KUKA KRL program: f1_Kuka_APT211T02S11.SRC

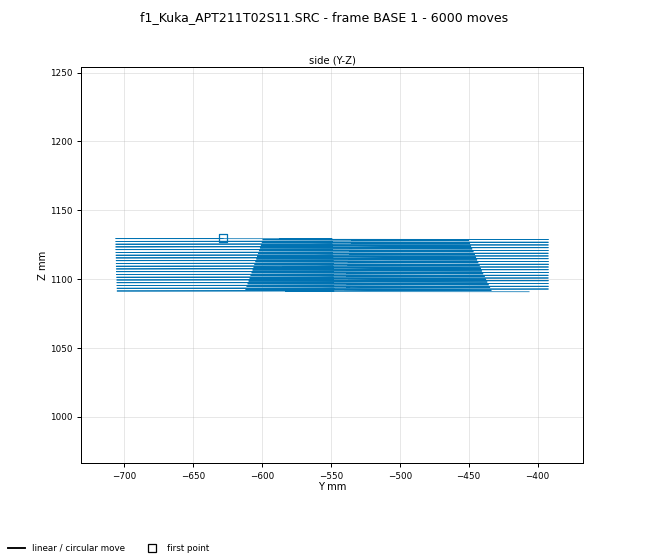
[picture p0: tool path of f1_Kuka_APT211T02S11.SRC in frame BASE 1, 6000 of 6001 moves have a stored position in this frame; points joined in program order, loops and branches not executed]
&ACCESS RVP
&REL 2
&PARAM TEMPLATE = C:\KRC\Roboter\Template\vorgabe
&PARAM EDITMASK = *
DEF f1_Kuka_APT211T02S11()


;FOLD INI;%{PE}%V3.2.0,%MKUKATPBASIS,%CINIT,%VCOMMON,%P
  ;FOLD BAS INI;%{E}%V3.2.0,%MKUKATPBASIS,%CINIT,%VINIT,%P
    GLOBAL INTERRUPT DECL 3 WHEN $STOPMESS==TRUE DO IR_STOPM ( )
    INTERRUPT ON 3
    BAS (#INITMOV,0 )
  ;ENDFOLD (BAS INI)
  ;FOLD USER INI;%{E}%V3.2.0,%MKUKATPUSER,%CINIT,%VINIT,%P
    ;Make your modifications here
  ;ENDFOLD (USER INI)
;ENDFOLD (INI)


;*** Make Null PTP Move
  PTP $pos_act

;*** Auto Load The Correct TOOL Data
  $tool=tool_data[2]

;*** Auto Load The Correct BASE Data
  $base=base_data[1]

  $ADVANCE = 5

;*** Restate Last Velocity
MMPM(30000.0)
SetRPM(8000)
LIN {X 0.276,Y -628.443,Z 1129.655,A 0.000,B 0.000,C 90.000,E1 153.896} C_DIS
LIN {X -0.160,Y -631.437,Z 1129.648,A 0.000,B 0.000,C 90.000,E1 152.666} C_DIS
LIN {X 0.011,Y -634.210,Z 1129.641,A 0.000,B 0.000,C 90.000,E1 151.385} C_DIS
LIN {X -0.027,Y -636.938,Z 1129.634,A 0.000,B 0.000,C 90.000,E1 150.127} C_DIS
LIN {X -0.018,Y -639.541,Z 1129.627,A 0.000,B 0.000,C 90.000,E1 148.869} C_DIS
LIN {X -0.027,Y -641.475,Z 1129.621,A 0.000,B 0.000,C 90.000,E1 147.867} C_DIS
LIN {X -0.154,Y -643.842,Z 1129.615,A 0.000,B 0.000,C 90.000,E1 146.628} C_DIS
LIN {X -0.238,Y -646.087,Z 1129.608,A 0.000,B 0.000,C 90.000,E1 145.388} C_DIS
LIN {X 0.084,Y -648.177,Z 1129.601,A 0.000,B 0.000,C 90.000,E1 144.116} C_DIS
LIN {X -0.031,Y -650.714,Z 1129.592,A 0.000,B 0.000,C 90.000,E1 142.637} C_DIS
LIN {X -0.300,Y -654.664,Z 1129.580,A 0.000,B 0.000,C 90.000,E1 140.436} C_DIS
LIN {X -0.032,Y -657.890,Z 1129.571,A 0.000,B 0.000,C 90.000,E1 138.690} C_DIS
LIN {X -0.154,Y -660.769,Z 1129.562,A 0.000,B 0.000,C 90.000,E1 137.229} C_DIS
LIN {X 0.211,Y -664.786,Z 1129.552,A 0.000,B 0.000,C 90.000,E1 135.243} C_DIS
LIN {X 0.204,Y -669.174,Z 1129.541,A 0.000,B 0.000,C 90.000,E1 133.299} C_DIS
LIN {X -0.116,Y -673.801,Z 1129.530,A 0.000,B 0.000,C 90.000,E1 131.391} C_DIS
LIN {X 0.050,Y -676.665,Z 1129.523,A 0.000,B 0.000,C 90.000,E1 130.172} C_DIS
LIN {X 0.038,Y -682.177,Z 1129.511,A 0.000,B 0.000,C 90.000,E1 128.016} C_DIS
LIN {X -0.141,Y -684.591,Z 1129.506,A 0.000,B 0.000,C 90.000,E1 127.076} C_DIS
LIN {X -0.113,Y -687.597,Z 1129.499,A 0.000,B 0.000,C 90.000,E1 125.884} C_DIS
LIN {X -0.232,Y -689.932,Z 1129.494,A 0.000,B 0.000,C 90.000,E1 124.945} C_DIS
LIN {X -0.261,Y -693.988,Z 1129.485,A 0.000,B 0.000,C 90.000,E1 123.293} C_DIS
LIN {X -0.123,Y -696.176,Z 1129.480,A 0.000,B 0.000,C 90.000,E1 122.339} C_DIS
LIN {X 0.292,Y -698.628,Z 1129.473,A 0.000,B 0.000,C 90.000,E1 121.131} C_DIS
LIN {X -0.135,Y -699.916,Z 1129.469,A 0.000,B 0.000,C 90.000,E1 120.463} C_DIS
LIN {X 0.203,Y -703.162,Z 1129.459,A 0.000,B 0.000,C 90.000,E1 118.565} C_DIS
LIN {X 0.147,Y -703.966,Z 1129.456,A 0.000,B 0.000,C 90.000,E1 118.103} C_DIS
LIN {X 0.378,Y -704.856,Z 1129.452,A 0.000,B 0.000,C 90.000,E1 117.385} C_DIS
LIN {X -0.043,Y -705.630,Z 1129.447,A 0.000,B 0.000,C 90.000,E1 116.488} C_DIS
LIN {X 0.182,Y -706.158,Z 1129.442,A 0.000,B 0.000,C 90.000,E1 115.540} C_DIS
LIN {X 0.128,Y -706.298,Z 1129.439,A 0.000,B 0.000,C 90.000,E1 115.079} C_DIS
LIN {X -0.226,Y -706.173,Z 1129.437,A 0.000,B 0.000,C 90.000,E1 114.643} C_DIS
LIN {X 0.066,Y -705.417,Z 1129.434,A 0.000,B 0.000,C 90.000,E1 114.155} C_DIS
LIN {X -0.288,Y -704.953,Z 1129.433,A 0.000,B 0.000,C 90.000,E1 113.951} C_DIS
LIN {X 0.000,Y -703.071,Z 1129.430,A 0.000,B 0.000,C 90.000,E1 113.462} C_DIS
LIN {X 0.281,Y -701.852,Z 1129.429,A 0.000,B 0.000,C 90.000,E1 113.206} C_DIS
LIN {X -0.094,Y -697.553,Z 1129.427,A 0.000,B 0.000,C 90.000,E1 112.770} C_DIS
LIN {X 0.035,Y -696.242,Z 1129.426,A 0.000,B 0.000,C 90.000,E1 112.642} C_DIS
LIN {X 0.163,Y -694.128,Z 1129.425,A 0.000,B 0.000,C 90.000,E1 112.514} C_DIS
LIN {X 0.381,Y -685.961,Z 1129.424,A 0.000,B 0.000,C 90.000,E1 112.206} C_DIS
LIN {X -0.097,Y -683.808,Z 1129.423,A 0.000,B 0.000,C 90.000,E1 112.206} C_DIS
LIN {X -0.315,Y -676.021,Z 1129.423,A 0.000,B 0.000,C 90.000,E1 112.153} C_DIS
LIN {X -0.314,Y -603.131,Z 1129.423,A 0.000,B 0.000,C 90.000,E1 112.153} C_DIS
LIN {X 0.332,Y -600.065,Z 1129.422,A 0.000,B 0.000,C 90.000,E1 111.897} C_DIS
LIN {X 0.084,Y -594.320,Z 1129.419,A 0.000,B 0.000,C 90.000,E1 111.461} C_DIS
LIN {X 0.254,Y -580.953,Z 1129.413,A 0.000,B 0.000,C 90.000,E1 110.248} C_DIS
LIN {X -0.197,Y -575.369,Z 1129.410,A 0.000,B 0.000,C 90.000,E1 109.812} C_DIS
LIN {X 0.116,Y -569.427,Z 1129.407,A 0.000,B 0.000,C 90.000,E1 109.322} C_DIS
LIN {X 0.032,Y -562.993,Z 1129.405,A 0.000,B 0.000,C 90.000,E1 108.906} C_DIS
LIN {X -0.161,Y -559.687,Z 1129.404,A 0.000,B 0.000,C 90.000,E1 108.725} C_DIS
LIN {X 0.065,Y -554.754,Z 1129.402,A 0.000,B 0.000,C 90.000,E1 108.417} C_DIS
LIN {X -0.112,Y -550.525,Z 1129.401,A 0.000,B 0.000,C 90.000,E1 108.109} C_DIS
LIN {X -0.149,Y -549.468,Z 1129.400,A 0.000,B 0.000,C 90.000,E1 107.928} C_DIS
LIN {X 0.332,Y -549.450,Z 1129.400,A 0.000,B 0.000,C 90.000,E1 107.873} C_DIS
LIN {X 0.089,Y -549.159,Z 1129.398,A 0.000,B 0.000,C 90.000,E1 107.583} C_DIS
LIN {X 0.132,Y -549.580,Z 1129.393,A 0.000,B 0.000,C 90.000,E1 106.677} C_DIS
LIN {X 0.156,Y -550.378,Z 1129.387,A 0.000,B 0.000,C 90.000,E1 105.552} C_DIS
LIN {X -0.172,Y -552.315,Z 1129.373,A 0.000,B 0.000,C 90.000,E1 103.063} C_DIS
LIN {X 0.140,Y -554.030,Z 1129.362,A 0.000,B 0.000,C 90.000,E1 101.074} C_DIS
LIN {X -0.191,Y -555.490,Z 1129.352,A 0.000,B 0.000,C 90.000,E1 99.434} C_DIS
LIN {X -0.135,Y -557.119,Z 1129.343,A 0.000,B 0.000,C 90.000,E1 97.757} C_DIS
LIN {X 0.026,Y -558.898,Z 1129.332,A 0.000,B 0.000,C 90.000,E1 95.796} C_DIS
LIN {X -0.037,Y -560.091,Z 1129.325,A 0.000,B 0.000,C 90.000,E1 94.416} C_DIS
LIN {X -0.085,Y -561.163,Z 1129.317,A 0.000,B 0.000,C 90.000,E1 93.037} C_DIS
LIN {X -0.149,Y -562.106,Z 1129.309,A 0.000,B 0.000,C 90.000,E1 91.661} C_DIS
LIN {X -0.001,Y -563.356,Z 1129.298,A 0.000,B 0.000,C 90.000,E1 89.714} C_DIS
LIN {X -0.039,Y -564.181,Z 1129.291,A 0.000,B 0.000,C 90.000,E1 88.339} C_DIS
LIN {X 0.194,Y -565.188,Z 1129.280,A 0.000,B 0.000,C 90.000,E1 86.388} C_DIS
LIN {X 0.242,Y -565.857,Z 1129.272,A 0.000,B 0.000,C 90.000,E1 85.008} C_DIS
LIN {X -0.005,Y -566.679,Z 1129.262,A 0.000,B 0.000,C 90.000,E1 83.109} C_DIS
LIN {X 0.122,Y -567.264,Z 1129.254,A 0.000,B 0.000,C 90.000,E1 81.724} C_DIS
LIN {X -0.041,Y -567.961,Z 1129.245,A 0.000,B 0.000,C 90.000,E1 80.095} C_DIS
LIN {X 0.175,Y -568.982,Z 1129.233,A 0.000,B 0.000,C 90.000,E1 77.881} C_DIS
LIN {X 0.105,Y -569.580,Z 1129.225,A 0.000,B 0.000,C 90.000,E1 76.520} C_DIS
LIN {X -0.317,Y -570.930,Z 1129.212,A 0.000,B 0.000,C 90.000,E1 74.102} C_DIS
LIN {X 0.136,Y -572.366,Z 1129.199,A 0.000,B 0.000,C 90.000,E1 71.873} C_DIS
LIN {X 0.092,Y -574.123,Z 1129.187,A 0.000,B 0.000,C 90.000,E1 69.699} C_DIS
LIN {X 0.119,Y -575.359,Z 1129.180,A 0.000,B 0.000,C 90.000,E1 68.337} C_DIS
LIN {X 0.174,Y -576.690,Z 1129.172,A 0.000,B 0.000,C 90.000,E1 66.975} C_DIS
LIN {X -0.052,Y -578.301,Z 1129.162,A 0.000,B 0.000,C 90.000,E1 65.101} C_DIS
LIN {X -0.246,Y -579.488,Z 1129.154,A 0.000,B 0.000,C 90.000,E1 63.768} C_DIS
LIN {X 0.216,Y -580.828,Z 1129.145,A 0.000,B 0.000,C 90.000,E1 62.103} C_DIS
LIN {X -0.041,Y -582.020,Z 1129.136,A 0.000,B 0.000,C 90.000,E1 60.511} C_DIS
LIN {X 0.213,Y -582.736,Z 1129.130,A 0.000,B 0.000,C 90.000,E1 59.410} C_DIS
LIN {X 0.297,Y -583.784,Z 1129.121,A 0.000,B 0.000,C 90.000,E1 57.788} C_DIS
LIN {X 0.096,Y -584.829,Z 1129.111,A 0.000,B 0.000,C 90.000,E1 55.928} C_DIS
LIN {X 0.169,Y -585.420,Z 1129.105,A 0.000,B 0.000,C 90.000,E1 54.848} C_DIS
LIN {X -0.150,Y -586.436,Z 1129.094,A 0.000,B 0.000,C 90.000,E1 53.004} C_DIS
LIN {X -0.115,Y -586.917,Z 1129.087,A 0.000,B 0.000,C 90.000,E1 51.662} C_DIS
LIN {X -0.170,Y -587.342,Z 1129.081,A 0.000,B 0.000,C 90.000,E1 50.598} C_DIS
LIN {X -0.117,Y -587.578,Z 1129.074,A 0.000,B 0.000,C 90.000,E1 49.256} C_DIS
LIN {X 0.137,Y -587.582,Z 1129.068,A 0.000,B 0.000,C 90.000,E1 48.162} C_DIS
LIN {X -0.099,Y -587.323,Z 1129.059,A 0.000,B 0.000,C 90.000,E1 46.581} C_DIS
LIN {X -0.090,Y -586.888,Z 1129.051,A 0.000,B 0.000,C 90.000,E1 45.243} C_DIS
LIN {X -0.262,Y -586.375,Z 1129.045,A 0.000,B 0.000,C 90.000,E1 44.190} C_DIS
LIN {X -0.191,Y -585.866,Z 1129.041,A 0.000,B 0.000,C 90.000,E1 43.380} C_DIS
LIN {X -0.272,Y -585.528,Z 1129.038,A 0.000,B 0.000,C 90.000,E1 42.852} C_DIS
LIN {X 0.133,Y -584.133,Z 1129.031,A 0.000,B 0.000,C 90.000,E1 41.472} C_DIS
LIN {X -0.042,Y -582.853,Z 1129.025,A 0.000,B 0.000,C 90.000,E1 40.415} C_DIS
LIN {X 0.040,Y -581.798,Z 1129.020,A 0.000,B 0.000,C 90.000,E1 39.600} C_DIS
LIN {X -0.170,Y -580.155,Z 1129.014,A 0.000,B 0.000,C 90.000,E1 38.543} C_DIS
LIN {X 0.204,Y -577.753,Z 1129.007,A 0.000,B 0.000,C 90.000,E1 37.156} C_DIS
LIN {X -0.125,Y -575.914,Z 1129.002,A 0.000,B 0.000,C 90.000,E1 36.377} C_DIS
LIN {X 0.331,Y -573.866,Z 1128.998,A 0.000,B 0.000,C 90.000,E1 35.518} C_DIS
LIN {X -0.179,Y -572.343,Z 1128.995,A 0.000,B 0.000,C 90.000,E1 35.025} C_DIS
LIN {X 0.035,Y -568.837,Z 1128.989,A 0.000,B 0.000,C 90.000,E1 33.913} C_DIS
LIN {X 0.082,Y -565.703,Z 1128.984,A 0.000,B 0.000,C 90.000,E1 33.086} C_DIS
LIN {X 0.094,Y -562.230,Z 1128.979,A 0.000,B 0.000,C 90.000,E1 32.260} C_DIS
LIN {X -0.212,Y -560.378,Z 1128.977,A 0.000,B 0.000,C 90.000,E1 31.878} C_DIS
LIN {X 0.213,Y -556.350,Z 1128.972,A 0.000,B 0.000,C 90.000,E1 31.003} C_DIS
LIN {X 0.057,Y -553.399,Z 1128.969,A 0.000,B 0.000,C 90.000,E1 30.463} C_DIS
LIN {X 0.121,Y -548.863,Z 1128.965,A 0.000,B 0.000,C 90.000,E1 29.617} C_DIS
LIN {X -0.212,Y -544.695,Z 1128.961,A 0.000,B 0.000,C 90.000,E1 28.949} C_DIS
LIN {X -0.107,Y -540.200,Z 1128.957,A 0.000,B 0.000,C 90.000,E1 28.231} C_DIS
LIN {X -0.044,Y -535.300,Z 1128.953,A 0.000,B 0.000,C 90.000,E1 27.513} C_DIS
LIN {X -0.032,Y -529.995,Z 1128.949,A 0.000,B 0.000,C 90.000,E1 26.796} C_DIS
LIN {X -0.151,Y -525.471,Z 1128.946,A 0.000,B 0.000,C 90.000,E1 26.232} C_DIS
LIN {X 0.118,Y -518.189,Z 1128.941,A 0.000,B 0.000,C 90.000,E1 25.335} C_DIS
LIN {X -0.146,Y -511.760,Z 1128.937,A 0.000,B 0.000,C 90.000,E1 24.643} C_DIS
LIN {X -0.046,Y -501.108,Z 1128.931,A 0.000,B 0.000,C 90.000,E1 23.515} C_DIS
LIN {X -0.219,Y -491.482,Z 1128.925,A 0.000,B 0.000,C 90.000,E1 22.589} C_DIS
LIN {X 0.230,Y -481.334,Z 1128.920,A 0.000,B 0.000,C 90.000,E1 21.589} C_DIS
LIN {X -0.214,Y -469.631,Z 1128.914,A 0.000,B 0.000,C 90.000,E1 20.610} C_DIS
LIN {X 0.057,Y -459.552,Z 1128.909,A 0.000,B 0.000,C 90.000,E1 19.685} C_DIS
LIN {X 0.000,Y -439.216,Z 1128.899,A 0.000,B 0.000,C 90.000,E1 17.819} C_DIS
LIN {X -0.060,Y -424.920,Z 1128.891,A 0.000,B 0.000,C 90.000,E1 16.370} C_DIS
LIN {X -0.192,Y -413.778,Z 1128.884,A 0.000,B 0.000,C 90.000,E1 15.134} C_DIS
LIN {X -0.059,Y -404.421,Z 1128.877,A 0.000,B 0.000,C 90.000,E1 13.939} C_DIS
LIN {X 0.035,Y -399.506,Z 1128.874,A 0.000,B 0.000,C 90.000,E1 13.244} C_DIS
LIN {X 0.011,Y -396.631,Z 1128.871,A 0.000,B 0.000,C 90.000,E1 12.771} C_DIS
LIN {X -0.041,Y -393.975,Z 1128.868,A 0.000,B 0.000,C 90.000,E1 12.187} C_DIS
LIN {X -0.016,Y -393.344,Z 1128.867,A 0.000,B 0.000,C 90.000,E1 12.007} C_DIS
LIN {X -0.132,Y -392.375,Z 1128.865,A 0.000,B 0.000,C 90.000,E1 11.658} C_DIS
LIN {X -0.158,Y -392.079,Z 1128.862,A 0.000,B 0.000,C 90.000,E1 11.130} C_DIS
LIN {X 0.147,Y -392.624,Z 1128.859,A 0.000,B 0.000,C 90.000,E1 10.546} C_DIS
LIN {X 0.104,Y -393.154,Z 1128.857,A 0.000,B 0.000,C 90.000,E1 10.197} C_DIS
LIN {X 0.021,Y -394.627,Z 1128.853,A 0.000,B 0.000,C 90.000,E1 9.500} C_DIS
LIN {X 0.161,Y -402.489,Z 1128.837,A 0.000,B 0.000,C 90.000,E1 6.663} C_DIS
LIN {X 0.143,Y -404.784,Z 1128.833,A 0.000,B 0.000,C 90.000,E1 5.967} C_DIS
LIN {X 0.033,Y -407.437,Z 1128.830,A 0.000,B 0.000,C 90.000,E1 5.391} C_DIS
LIN {X -0.183,Y -411.799,Z 1128.827,A 0.000,B 0.000,C 90.000,E1 4.816} C_DIS
LIN {X -0.014,Y -417.173,Z 1128.824,A 0.000,B 0.000,C 90.000,E1 4.359} C_DIS
LIN {X 0.006,Y -434.964,Z 1128.817,A 0.000,B 0.000,C 90.000,E1 3.094} C_DIS
LIN {X 0.033,Y -459.488,Z 1128.808,A 0.000,B 0.000,C 90.000,E1 1.432} C_DIS
LIN {X -0.093,Y -467.649,Z 1128.805,A 0.000,B 0.000,C 90.000,E1 0.917} C_DIS
LIN {X -0.004,Y -478.874,Z 1128.801,A 0.000,B 0.000,C 90.000,E1 0.172} C_DIS
LIN {X -0.194,Y -489.209,Z 1128.797,A 0.000,B 0.000,C 90.000,E1 359.484} C_DIS
LIN {X -0.158,Y -498.343,Z 1128.793,A 0.000,B 0.000,C 90.000,E1 358.797} C_DIS
LIN {X -0.226,Y -502.919,Z 1128.791,A 0.000,B 0.000,C 90.000,E1 358.453} C_DIS
LIN {X -0.004,Y -510.065,Z 1128.788,A 0.000,B 0.000,C 90.000,E1 357.822} C_DIS
LIN {X -0.067,Y -517.099,Z 1128.784,A 0.000,B 0.000,C 90.000,E1 357.192} C_DIS
LIN {X -0.231,Y -522.381,Z 1128.781,A 0.000,B 0.000,C 90.000,E1 356.674} C_DIS
LIN {X 0.171,Y -526.361,Z 1128.779,A 0.000,B 0.000,C 90.000,E1 356.216} C_DIS
LIN {X -0.037,Y -532.551,Z 1128.775,A 0.000,B 0.000,C 90.000,E1 355.527} C_DIS
LIN {X 0.238,Y -538.039,Z 1128.771,A 0.000,B 0.000,C 90.000,E1 354.780} C_DIS
LIN {X -0.248,Y -542.168,Z 1128.768,A 0.000,B 0.000,C 90.000,E1 354.261} C_DIS
LIN {X 0.111,Y -546.634,Z 1128.764,A 0.000,B 0.000,C 90.000,E1 353.514} C_DIS
LIN {X 0.035,Y -550.776,Z 1128.760,A 0.000,B 0.000,C 90.000,E1 352.818} C_DIS
LIN {X 0.179,Y -553.798,Z 1128.757,A 0.000,B 0.000,C 90.000,E1 352.243} C_DIS
LIN {X -0.209,Y -556.605,Z 1128.754,A 0.000,B 0.000,C 90.000,E1 351.724} C_DIS
LIN {X -0.196,Y -559.702,Z 1128.750,A 0.000,B 0.000,C 90.000,E1 351.027} C_DIS
LIN {X 0.245,Y -563.057,Z 1128.745,A 0.000,B 0.000,C 90.000,E1 350.151} C_DIS
LIN {X -0.093,Y -565.111,Z 1128.742,A 0.000,B 0.000,C 90.000,E1 349.634} C_DIS
LIN {X -0.147,Y -568.067,Z 1128.738,A 0.000,B 0.000,C 90.000,E1 348.814} C_DIS
LIN {X 0.021,Y -571.609,Z 1128.732,A 0.000,B 0.000,C 90.000,E1 347.701} C_DIS
LIN {X 0.238,Y -574.908,Z 1128.726,A 0.000,B 0.000,C 90.000,E1 346.589} C_DIS
LIN {X 0.077,Y -577.993,Z 1128.720,A 0.000,B 0.000,C 90.000,E1 345.519} C_DIS
LIN {X 0.183,Y -581.645,Z 1128.712,A 0.000,B 0.000,C 90.000,E1 344.157} C_DIS
LIN {X -0.108,Y -583.762,Z 1128.708,A 0.000,B 0.000,C 90.000,E1 343.378} C_DIS
LIN {X 0.259,Y -587.109,Z 1128.700,A 0.000,B 0.000,C 90.000,E1 342.000} C_DIS
LIN {X -0.114,Y -589.570,Z 1128.694,A 0.000,B 0.000,C 90.000,E1 340.967} C_DIS
LIN {X 0.102,Y -591.882,Z 1128.688,A 0.000,B 0.000,C 90.000,E1 339.880} C_DIS
LIN {X 0.232,Y -594.457,Z 1128.681,A 0.000,B 0.000,C 90.000,E1 338.539} C_DIS
LIN {X 0.030,Y -595.433,Z 1128.678,A 0.000,B 0.000,C 90.000,E1 338.028} C_DIS
LIN {X 0.071,Y -596.576,Z 1128.674,A 0.000,B 0.000,C 90.000,E1 337.230} C_DIS
LIN {X -0.053,Y -598.137,Z 1128.666,A 0.000,B 0.000,C 90.000,E1 335.921} C_DIS
LIN {X 0.173,Y -599.005,Z 1128.660,A 0.000,B 0.000,C 90.000,E1 334.845} C_DIS
LIN {X -0.054,Y -599.388,Z 1128.656,A 0.000,B 0.000,C 90.000,E1 334.076} C_DIS
LIN {X 0.262,Y -599.490,Z 1128.652,A 0.000,B 0.000,C 90.000,E1 333.256} C_DIS
LIN {X -0.037,Y -599.218,Z 1128.646,A 0.000,B 0.000,C 90.000,E1 332.231} C_DIS
LIN {X 0.018,Y -598.634,Z 1128.641,A 0.000,B 0.000,C 90.000,E1 331.435} C_DIS
LIN {X -0.139,Y -598.037,Z 1128.638,A 0.000,B 0.000,C 90.000,E1 330.923} C_DIS
LIN {X -0.092,Y -596.865,Z 1128.634,A 0.000,B 0.000,C 90.000,E1 330.127} C_DIS
LIN {X -0.055,Y -595.245,Z 1128.630,A 0.000,B 0.000,C 90.000,E1 329.331} C_DIS
LIN {X -0.037,Y -593.230,Z 1128.625,A 0.000,B 0.000,C 90.000,E1 328.535} C_DIS
LIN {X -0.141,Y -592.478,Z 1128.624,A 0.000,B 0.000,C 90.000,E1 328.280} C_DIS
LIN {X 0.156,Y -589.637,Z 1128.619,A 0.000,B 0.000,C 90.000,E1 327.454} C_DIS
LIN {X -0.386,Y -586.404,Z 1128.615,A 0.000,B 0.000,C 90.000,E1 326.707} C_DIS
LIN {X -0.076,Y -583.355,Z 1128.611,A 0.000,B 0.000,C 90.000,E1 326.008} C_DIS
LIN {X 0.202,Y -579.925,Z 1128.607,A 0.000,B 0.000,C 90.000,E1 325.308} C_DIS
LIN {X 0.201,Y -576.931,Z 1128.604,A 0.000,B 0.000,C 90.000,E1 324.769} C_DIS
LIN {X -0.006,Y -570.210,Z 1128.598,A 0.000,B 0.000,C 90.000,E1 323.703} C_DIS
LIN {X 0.159,Y -565.536,Z 1128.595,A 0.000,B 0.000,C 90.000,E1 323.004} C_DIS
LIN {X -0.095,Y -557.371,Z 1128.589,A 0.000,B 0.000,C 90.000,E1 321.949} C_DIS
LIN {X 0.062,Y -549.505,Z 1128.583,A 0.000,B 0.000,C 90.000,E1 320.964} C_DIS
LIN {X 0.174,Y -537.721,Z 1128.575,A 0.000,B 0.000,C 90.000,E1 319.542} C_DIS
LIN {X -0.223,Y -535.682,Z 1128.574,A 0.000,B 0.000,C 90.000,E1 319.299} C_DIS
LIN {X 0.123,Y -532.461,Z 1128.571,A 0.000,B 0.000,C 90.000,E1 318.690} C_DIS
LIN {X -0.060,Y -531.568,Z 1128.570,A 0.000,B 0.000,C 90.000,E1 318.566} C_DIS
LIN {X 0.109,Y -530.858,Z 1128.569,A 0.000,B 0.000,C 90.000,E1 318.405} C_DIS
LIN {X -0.199,Y -530.175,Z 1128.568,A 0.000,B 0.000,C 90.000,E1 318.243} C_DIS
LIN {X -0.059,Y -528.452,Z 1128.566,A 0.000,B 0.000,C 90.000,E1 317.796} C_DIS
LIN {X -0.160,Y -526.830,Z 1128.562,A 0.000,B 0.000,C 90.000,E1 317.229} C_DIS
LIN {X -0.043,Y -526.104,Z 1128.560,A 0.000,B 0.000,C 90.000,E1 316.782} C_DIS
LIN {X 0.155,Y -525.395,Z 1128.555,A 0.000,B 0.000,C 90.000,E1 315.891} C_DIS
LIN {X 0.037,Y -525.202,Z 1128.552,A 0.000,B 0.000,C 90.000,E1 315.324} C_DIS
LIN {X 0.105,Y -524.824,Z 1128.544,A 0.000,B 0.000,C 90.000,E1 313.866} C_DIS
LIN {X -0.117,Y -525.254,Z 1128.528,A 0.000,B 0.000,C 90.000,E1 310.987} C_DIS
LIN {X -0.140,Y -526.429,Z 1128.515,A 0.000,B 0.000,C 90.000,E1 308.669} C_DIS
LIN {X 0.003,Y -527.504,Z 1128.505,A 0.000,B 0.000,C 90.000,E1 306.916} C_DIS
LIN {X -0.032,Y -528.643,Z 1128.495,A 0.000,B 0.000,C 90.000,E1 305.185} C_DIS
LIN {X -0.126,Y -529.510,Z 1128.489,A 0.000,B 0.000,C 90.000,E1 304.040} C_DIS
LIN {X 0.022,Y -530.997,Z 1128.478,A 0.000,B 0.000,C 90.000,E1 302.005} C_DIS
LIN {X 0.229,Y -532.317,Z 1128.468,A 0.000,B 0.000,C 90.000,E1 300.256} C_DIS
LIN {X 0.044,Y -533.168,Z 1128.462,A 0.000,B 0.000,C 90.000,E1 299.127} C_DIS
LIN {X 0.083,Y -533.934,Z 1128.456,A 0.000,B 0.000,C 90.000,E1 297.975} C_DIS
LIN {X 0.144,Y -534.499,Z 1128.449,A 0.000,B 0.000,C 90.000,E1 296.821} C_DIS
LIN {X -0.269,Y -534.874,Z 1128.443,A 0.000,B 0.000,C 90.000,E1 295.720} C_DIS
LIN {X 0.281,Y -534.998,Z 1128.436,A 0.000,B 0.000,C 90.000,E1 294.515} C_DIS
LIN {X 0.124,Y -535.054,Z 1128.430,A 0.000,B 0.000,C 90.000,E1 293.387} C_DIS
LIN {X -0.031,Y -535.106,Z 1128.422,A 0.000,B 0.000,C 90.000,E1 291.972} C_DIS
LIN {X 0.028,Y -534.993,Z 1128.413,A 0.000,B 0.000,C 90.000,E1 290.248} C_DIS
LIN {X -0.137,Y -534.782,Z 1128.405,A 0.000,B 0.000,C 90.000,E1 288.833} C_DIS
LIN {X -0.144,Y -534.430,Z 1128.397,A 0.000,B 0.000,C 90.000,E1 287.402} C_DIS
LIN {X -0.186,Y -534.064,Z 1128.390,A 0.000,B 0.000,C 90.000,E1 286.260} C_DIS
LIN {X -0.158,Y -533.295,Z 1128.381,A 0.000,B 0.000,C 90.000,E1 284.537} C_DIS
LIN {X 0.194,Y -532.589,Z 1128.373,A 0.000,B 0.000,C 90.000,E1 283.063} C_DIS
LIN {X -0.056,Y -531.688,Z 1128.363,A 0.000,B 0.000,C 90.000,E1 281.366} C_DIS
LIN {X 0.191,Y -530.743,Z 1128.354,A 0.000,B 0.000,C 90.000,E1 279.613} C_DIS
LIN {X -0.280,Y -529.834,Z 1128.344,A 0.000,B 0.000,C 90.000,E1 277.936} C_DIS
LIN {X -0.223,Y -528.819,Z 1128.333,A 0.000,B 0.000,C 90.000,E1 275.910} C_DIS
LIN {X 0.236,Y -528.209,Z 1128.325,A 0.000,B 0.000,C 90.000,E1 274.416} C_DIS
LIN {X 0.156,Y -527.568,Z 1128.317,A 0.000,B 0.000,C 90.000,E1 272.980} C_DIS
LIN {X 0.004,Y -526.806,Z 1128.307,A 0.000,B 0.000,C 90.000,E1 271.260} C_DIS
LIN {X -0.171,Y -525.989,Z 1128.297,A 0.000,B 0.000,C 90.000,E1 269.542} C_DIS
LIN {X 0.225,Y -525.480,Z 1128.291,A 0.000,B 0.000,C 90.000,E1 268.339} C_DIS
LIN {X 0.061,Y -524.748,Z 1128.283,A 0.000,B 0.000,C 90.000,E1 266.906} C_DIS
LIN {X -0.086,Y -523.713,Z 1128.273,A 0.000,B 0.000,C 90.000,E1 265.179} C_DIS
LIN {X -0.241,Y -522.938,Z 1128.267,A 0.000,B 0.000,C 90.000,E1 264.033} C_DIS
LIN {X 0.150,Y -521.520,Z 1128.259,A 0.000,B 0.000,C 90.000,E1 262.534} C_DIS
LIN {X 0.071,Y -520.126,Z 1128.251,A 0.000,B 0.000,C 90.000,E1 261.084} C_DIS
LIN {X -0.033,Y -518.715,Z 1128.242,A 0.000,B 0.000,C 90.000,E1 259.634} C_DIS
LIN {X -0.071,Y -517.334,Z 1128.234,A 0.000,B 0.000,C 90.000,E1 258.173} C_DIS
LIN {X -0.057,Y -515.314,Z 1128.223,A 0.000,B 0.000,C 90.000,E1 256.117} C_DIS
LIN {X 0.085,Y -514.002,Z 1128.215,A 0.000,B 0.000,C 90.000,E1 254.629} C_DIS
LIN {X 0.165,Y -512.216,Z 1128.205,A 0.000,B 0.000,C 90.000,E1 252.851} C_DIS
LIN {X -0.041,Y -511.026,Z 1128.198,A 0.000,B 0.000,C 90.000,E1 251.692} C_DIS
LIN {X 0.061,Y -509.782,Z 1128.192,A 0.000,B 0.000,C 90.000,E1 250.496} C_DIS
LIN {X -0.071,Y -508.118,Z 1128.183,A 0.000,B 0.000,C 90.000,E1 249.028} C_DIS
LIN {X -0.045,Y -506.433,Z 1128.175,A 0.000,B 0.000,C 90.000,E1 247.539} C_DIS
LIN {X -0.136,Y -504.926,Z 1128.169,A 0.000,B 0.000,C 90.000,E1 246.357} C_DIS
LIN {X -0.045,Y -503.360,Z 1128.162,A 0.000,B 0.000,C 90.000,E1 245.153} C_DIS
LIN {X 0.096,Y -501.199,Z 1128.154,A 0.000,B 0.000,C 90.000,E1 243.640} C_DIS
LIN {X 0.123,Y -499.434,Z 1128.147,A 0.000,B 0.000,C 90.000,E1 242.436} C_DIS
LIN {X 0.191,Y -497.098,Z 1128.139,A 0.000,B 0.000,C 90.000,E1 240.923} C_DIS
LIN {X 0.219,Y -494.663,Z 1128.130,A 0.000,B 0.000,C 90.000,E1 239.410} C_DIS
LIN {X 0.293,Y -491.602,Z 1128.120,A 0.000,B 0.000,C 90.000,E1 237.582} C_DIS
LIN {X 0.051,Y -489.060,Z 1128.112,A 0.000,B 0.000,C 90.000,E1 236.087} C_DIS
LIN {X -0.140,Y -485.944,Z 1128.101,A 0.000,B 0.000,C 90.000,E1 234.276} C_DIS
LIN {X 0.057,Y -483.240,Z 1128.093,A 0.000,B 0.000,C 90.000,E1 232.718} C_DIS
LIN {X 0.001,Y -481.107,Z 1128.086,A 0.000,B 0.000,C 90.000,E1 231.492} C_DIS
LIN {X 0.120,Y -477.710,Z 1128.076,A 0.000,B 0.000,C 90.000,E1 229.622} C_DIS
LIN {X 0.121,Y -474.327,Z 1128.065,A 0.000,B 0.000,C 90.000,E1 227.757} C_DIS
LIN {X 0.139,Y -470.398,Z 1128.053,A 0.000,B 0.000,C 90.000,E1 225.567} C_DIS
LIN {X -0.141,Y -465.834,Z 1128.038,A 0.000,B 0.000,C 90.000,E1 222.771} C_DIS
LIN {X 0.043,Y -462.152,Z 1128.024,A 0.000,B 0.000,C 90.000,E1 220.216} C_DIS
LIN {X 0.093,Y -459.617,Z 1128.013,A 0.000,B 0.000,C 90.000,E1 218.302} C_DIS
LIN {X -0.095,Y -457.023,Z 1128.000,A 0.000,B 0.000,C 90.000,E1 216.091} C_DIS
LIN {X 0.295,Y -454.845,Z 1127.990,A 0.000,B 0.000,C 90.000,E1 214.119} C_DIS
LIN {X 0.202,Y -451.679,Z 1127.970,A 0.000,B 0.000,C 90.000,E1 210.590} C_DIS
LIN {X -0.051,Y -449.938,Z 1127.949,A 0.000,B 0.000,C 90.000,E1 206.744} C_DIS
LIN {X -0.278,Y -450.279,Z 1127.940,A 0.000,B 0.000,C 90.000,E1 205.155} C_DIS
LIN {X 0.027,Y -451.189,Z 1127.932,A 0.000,B 0.000,C 90.000,E1 203.823} C_DIS
LIN {X 0.099,Y -452.383,Z 1127.927,A 0.000,B 0.000,C 90.000,E1 202.845} C_DIS
LIN {X 0.056,Y -455.799,Z 1127.916,A 0.000,B 0.000,C 90.000,E1 200.918} C_DIS
LIN {X 0.005,Y -459.488,Z 1127.907,A 0.000,B 0.000,C 90.000,E1 199.322} C_DIS
LIN {X 0.017,Y -466.025,Z 1127.895,A 0.000,B 0.000,C 90.000,E1 197.094} C_DIS
LIN {X -0.103,Y -474.605,Z 1127.881,A 0.000,B 0.000,C 90.000,E1 194.592} C_DIS
LIN {X 0.013,Y -486.289,Z 1127.864,A 0.000,B 0.000,C 90.000,E1 191.478} C_DIS
LIN {X 0.194,Y -494.854,Z 1127.852,A 0.000,B 0.000,C 90.000,E1 189.321} C_DIS
LIN {X 0.168,Y -501.028,Z 1127.844,A 0.000,B 0.000,C 90.000,E1 187.814} C_DIS
LIN {X -0.247,Y -505.941,Z 1127.837,A 0.000,B 0.000,C 90.000,E1 186.663} C_DIS
LIN {X -0.138,Y -511.919,Z 1127.829,A 0.000,B 0.000,C 90.000,E1 185.163} C_DIS
LIN {X 0.113,Y -516.758,Z 1127.822,A 0.000,B 0.000,C 90.000,E1 183.955} C_DIS
LIN {X -0.219,Y -524.051,Z 1127.812,A 0.000,B 0.000,C 90.000,E1 182.236} C_DIS
LIN {X -0.140,Y -531.802,Z 1127.802,A 0.000,B 0.000,C 90.000,E1 180.344} C_DIS
LIN {X -0.164,Y -536.667,Z 1127.796,A 0.000,B 0.000,C 90.000,E1 179.198} C_DIS
LIN {X 0.195,Y -543.296,Z 1127.787,A 0.000,B 0.000,C 90.000,E1 177.593} C_DIS
LIN {X 0.228,Y -551.080,Z 1127.777,A 0.000,B 0.000,C 90.000,E1 175.755} C_DIS
LIN {X -0.065,Y -558.889,Z 1127.766,A 0.000,B 0.000,C 90.000,E1 173.970} C_DIS
LIN {X 0.209,Y -567.288,Z 1127.756,A 0.000,B 0.000,C 90.000,E1 172.008} C_DIS
LIN {X 0.000,Y -574.375,Z 1127.747,A 0.000,B 0.000,C 90.000,E1 170.387} C_DIS
LIN {X -0.198,Y -580.103,Z 1127.739,A 0.000,B 0.000,C 90.000,E1 169.050} C_DIS
LIN {X -0.190,Y -585.565,Z 1127.732,A 0.000,B 0.000,C 90.000,E1 167.701} C_DIS
LIN {X -0.085,Y -590.948,Z 1127.724,A 0.000,B 0.000,C 90.000,E1 166.353} C_DIS
LIN {X 0.252,Y -596.015,Z 1127.717,A 0.000,B 0.000,C 90.000,E1 164.991} C_DIS
LIN {X 0.103,Y -598.873,Z 1127.712,A 0.000,B 0.000,C 90.000,E1 164.212} C_DIS
LIN {X 0.282,Y -602.430,Z 1127.707,A 0.000,B 0.000,C 90.000,E1 163.142} C_DIS
LIN {X -0.161,Y -606.719,Z 1127.699,A 0.000,B 0.000,C 90.000,E1 161.873} C_DIS
LIN {X 0.042,Y -610.721,Z 1127.692,A 0.000,B 0.000,C 90.000,E1 160.550} C_DIS
LIN {X -0.017,Y -613.792,Z 1127.686,A 0.000,B 0.000,C 90.000,E1 159.518} C_DIS
LIN {X -0.075,Y -617.327,Z 1127.679,A 0.000,B 0.000,C 90.000,E1 158.230} C_DIS
LIN {X 0.151,Y -621.444,Z 1127.671,A 0.000,B 0.000,C 90.000,E1 156.666} C_DIS
LIN {X -0.105,Y -624.680,Z 1127.663,A 0.000,B 0.000,C 90.000,E1 155.409} C_DIS
LIN {X -0.314,Y -627.838,Z 1127.656,A 0.000,B 0.000,C 90.000,E1 154.152} C_DIS
LIN {X -0.202,Y -630.870,Z 1127.649,A 0.000,B 0.000,C 90.000,E1 152.871} C_DIS
LIN {X -0.111,Y -632.572,Z 1127.645,A 0.000,B 0.000,C 90.000,E1 152.103} C_DIS
LIN {X -0.138,Y -635.866,Z 1127.637,A 0.000,B 0.000,C 90.000,E1 150.589} C_DIS
LIN {X -0.147,Y -638.504,Z 1127.630,A 0.000,B 0.000,C 90.000,E1 149.331} C_DIS
LIN {X -0.167,Y -640.540,Z 1127.624,A 0.000,B 0.000,C 90.000,E1 148.329} C_DIS
LIN {X -0.253,Y -643.369,Z 1127.616,A 0.000,B 0.000,C 90.000,E1 146.834} C_DIS
LIN {X -0.346,Y -645.624,Z 1127.609,A 0.000,B 0.000,C 90.000,E1 145.595} C_DIS
LIN {X -0.031,Y -647.756,Z 1127.602,A 0.000,B 0.000,C 90.000,E1 144.322} C_DIS
LIN {X -0.150,Y -650.297,Z 1127.594,A 0.000,B 0.000,C 90.000,E1 142.844} C_DIS
LIN {X 0.080,Y -654.237,Z 1127.581,A 0.000,B 0.000,C 90.000,E1 140.598} C_DIS
LIN {X -0.123,Y -656.980,Z 1127.573,A 0.000,B 0.000,C 90.000,E1 139.138} C_DIS
LIN {X 0.203,Y -660.334,Z 1127.563,A 0.000,B 0.000,C 90.000,E1 137.391} C_DIS
LIN {X 0.079,Y -664.818,Z 1127.551,A 0.000,B 0.000,C 90.000,E1 135.202} C_DIS
LIN {X 0.092,Y -669.805,Z 1127.539,A 0.000,B 0.000,C 90.000,E1 133.014} C_DIS
LIN {X 0.226,Y -673.866,Z 1127.530,A 0.000,B 0.000,C 90.000,E1 131.310} C_DIS
LIN {X 0.392,Y -676.737,Z 1127.523,A 0.000,B 0.000,C 90.000,E1 130.092} C_DIS
LIN {X -0.037,Y -682.266,Z 1127.511,A 0.000,B 0.000,C 90.000,E1 127.971} C_DIS
LIN {X 0.175,Y -684.128,Z 1127.507,A 0.000,B 0.000,C 90.000,E1 127.237} C_DIS
LIN {X 0.231,Y -687.671,Z 1127.499,A 0.000,B 0.000,C 90.000,E1 125.804} C_DIS
LIN {X 0.313,Y -690.589,Z 1127.492,A 0.000,B 0.000,C 90.000,E1 124.612} C_DIS
LIN {X 0.081,Y -694.062,Z 1127.485,A 0.000,B 0.000,C 90.000,E1 123.214} C_DIS
LIN {X -0.154,Y -696.246,Z 1127.479,A 0.000,B 0.000,C 90.000,E1 122.291} C_DIS
LIN {X 0.016,Y -698.267,Z 1127.474,A 0.000,B 0.000,C 90.000,E1 121.337} C_DIS
LIN {X 0.202,Y -700.000,Z 1127.469,A 0.000,B 0.000,C 90.000,E1 120.384} C_DIS
LIN {X -0.082,Y -703.222,Z 1127.458,A 0.000,B 0.000,C 90.000,E1 118.537} C_DIS
LIN {X 0.146,Y -704.000,Z 1127.456,A 0.000,B 0.000,C 90.000,E1 118.052} C_DIS
LIN {X -0.244,Y -704.865,Z 1127.452,A 0.000,B 0.000,C 90.000,E1 117.385} C_DIS
LIN {X -0.008,Y -705.447,Z 1127.448,A 0.000,B 0.000,C 90.000,E1 116.668} C_DIS
LIN {X 0.209,Y -706.066,Z 1127.443,A 0.000,B 0.000,C 90.000,E1 115.720} C_DIS
LIN {X -0.148,Y -706.260,Z 1127.440,A 0.000,B 0.000,C 90.000,E1 115.283} C_DIS
LIN {X -0.207,Y -706.127,Z 1127.437,A 0.000,B 0.000,C 90.000,E1 114.591} C_DIS
LIN {X 0.376,Y -705.321,Z 1127.434,A 0.000,B 0.000,C 90.000,E1 114.079} C_DIS
LIN {X -0.267,Y -704.779,Z 1127.433,A 0.000,B 0.000,C 90.000,E1 113.898} C_DIS
LIN {X 0.303,Y -702.866,Z 1127.430,A 0.000,B 0.000,C 90.000,E1 113.387} C_DIS
LIN {X 0.165,Y -702.299,Z 1127.429,A 0.000,B 0.000,C 90.000,E1 113.281} C_DIS
LIN {X -0.340,Y -701.434,Z 1127.429,A 0.000,B 0.000,C 90.000,E1 113.206} C_DIS
LIN {X -0.073,Y -697.047,Z 1127.426,A 0.000,B 0.000,C 90.000,E1 112.717} C_DIS
LIN {X 0.057,Y -695.464,Z 1127.426,A 0.000,B 0.000,C 90.000,E1 112.589} C_DIS
LIN {X 0.184,Y -692.717,Z 1127.425,A 0.000,B 0.000,C 90.000,E1 112.461} C_DIS
LIN {X -0.027,Y -687.201,Z 1127.424,A 0.000,B 0.000,C 90.000,E1 112.280} C_DIS
LIN {X 0.167,Y -685.346,Z 1127.423,A 0.000,B 0.000,C 90.000,E1 112.206} C_DIS
LIN {X -0.287,Y -682.525,Z 1127.423,A 0.000,B 0.000,C 90.000,E1 112.206} C_DIS
LIN {X -0.335,Y -676.711,Z 1127.423,A 0.000,B 0.000,C 90.000,E1 112.153} C_DIS
LIN {X -0.346,Y -603.224,Z 1127.423,A 0.000,B 0.000,C 90.000,E1 112.153} C_DIS
LIN {X 0.242,Y -600.029,Z 1127.422,A 0.000,B 0.000,C 90.000,E1 111.897} C_DIS
LIN {X 0.129,Y -594.412,Z 1127.419,A 0.000,B 0.000,C 90.000,E1 111.461} C_DIS
LIN {X -0.048,Y -579.760,Z 1127.412,A 0.000,B 0.000,C 90.000,E1 110.174} C_DIS
LIN {X 0.055,Y -574.077,Z 1127.409,A 0.000,B 0.000,C 90.000,E1 109.685} C_DIS
LIN {X 0.226,Y -568.072,Z 1127.407,A 0.000,B 0.000,C 90.000,E1 109.214} C_DIS
LIN {X -0.125,Y -561.634,Z 1127.405,A 0.000,B 0.000,C 90.000,E1 108.833} C_DIS
LIN {X 0.165,Y -554.932,Z 1127.402,A 0.000,B 0.000,C 90.000,E1 108.417} C_DIS
LIN {X -0.070,Y -550.438,Z 1127.401,A 0.000,B 0.000,C 90.000,E1 108.109} C_DIS
LIN {X -0.103,Y -549.383,Z 1127.400,A 0.000,B 0.000,C 90.000,E1 107.928} C_DIS
LIN {X -0.145,Y -549.366,Z 1127.400,A 0.000,B 0.000,C 90.000,E1 107.928} C_DIS
LIN {X -0.187,Y -549.073,Z 1127.397,A 0.000,B 0.000,C 90.000,E1 107.511} C_DIS
LIN {X 0.097,Y -550.262,Z 1127.387,A 0.000,B 0.000,C 90.000,E1 105.607} C_DIS
LIN {X -0.240,Y -552.183,Z 1127.373,A 0.000,B 0.000,C 90.000,E1 103.119} C_DIS
LIN {X 0.064,Y -553.894,Z 1127.362,A 0.000,B 0.000,C 90.000,E1 101.130} C_DIS
LIN {X 0.184,Y -555.382,Z 1127.353,A 0.000,B 0.000,C 90.000,E1 99.443} C_DIS
LIN {X -0.166,Y -557.248,Z 1127.342,A 0.000,B 0.000,C 90.000,E1 97.530} C_DIS
LIN {X 0.007,Y -559.065,Z 1127.331,A 0.000,B 0.000,C 90.000,E1 95.568} C_DIS
LIN {X -0.048,Y -560.243,Z 1127.323,A 0.000,B 0.000,C 90.000,E1 94.188} C_DIS
LIN {X -0.090,Y -561.300,Z 1127.316,A 0.000,B 0.000,C 90.000,E1 92.808} C_DIS
LIN {X -0.150,Y -562.227,Z 1127.308,A 0.000,B 0.000,C 90.000,E1 91.432} C_DIS
LIN {X 0.002,Y -563.445,Z 1127.297,A 0.000,B 0.000,C 90.000,E1 89.484} C_DIS
LIN {X 0.089,Y -564.376,Z 1127.288,A 0.000,B 0.000,C 90.000,E1 87.822} C_DIS
LIN {X -0.225,Y -565.354,Z 1127.277,A 0.000,B 0.000,C 90.000,E1 85.927} C_DIS
LIN {X -0.170,Y -565.959,Z 1127.270,A 0.000,B 0.000,C 90.000,E1 84.546} C_DIS
LIN {X 0.148,Y -566.791,Z 1127.259,A 0.000,B 0.000,C 90.000,E1 82.591} C_DIS
LIN {X 0.014,Y -567.139,Z 1127.254,A 0.000,B 0.000,C 90.000,E1 81.781} C_DIS
LIN {X -0.150,Y -567.826,Z 1127.245,A 0.000,B 0.000,C 90.000,E1 80.151} C_DIS
LIN {X 0.066,Y -568.817,Z 1127.233,A 0.000,B 0.000,C 90.000,E1 77.937} C_DIS
LIN {X -0.137,Y -569.434,Z 1127.225,A 0.000,B 0.000,C 90.000,E1 76.589} C_DIS
LIN {X 0.314,Y -570.407,Z 1127.215,A 0.000,B 0.000,C 90.000,E1 74.629} C_DIS
LIN {X 0.093,Y -571.099,Z 1127.209,A 0.000,B 0.000,C 90.000,E1 73.559} C_DIS
LIN {X -0.166,Y -572.641,Z 1127.197,A 0.000,B 0.000,C 90.000,E1 71.402} C_DIS
LIN {X -0.188,Y -574.745,Z 1127.183,A 0.000,B 0.000,C 90.000,E1 68.954} C_DIS
LIN {X -0.150,Y -576.534,Z 1127.172,A 0.000,B 0.000,C 90.000,E1 67.050} C_DIS
LIN {X 0.148,Y -577.650,Z 1127.165,A 0.000,B 0.000,C 90.000,E1 65.665} C_DIS
LIN {X -0.055,Y -578.862,Z 1127.157,A 0.000,B 0.000,C 90.000,E1 64.332} C_DIS
LIN {X -0.239,Y -580.000,Z 1127.150,A 0.000,B 0.000,C 90.000,E1 62.999} C_DIS
LIN {X -0.146,Y -581.063,Z 1127.142,A 0.000,B 0.000,C 90.000,E1 61.641} C_DIS
LIN {X 0.111,Y -582.229,Z 1127.133,A 0.000,B 0.000,C 90.000,E1 59.999} C_DIS
LIN {X 0.050,Y -583.424,Z 1127.123,A 0.000,B 0.000,C 90.000,E1 58.122} C_DIS
LIN {X 0.329,Y -584.479,Z 1127.113,A 0.000,B 0.000,C 90.000,E1 56.215} C_DIS
LIN {X 0.102,Y -585.213,Z 1127.105,A 0.000,B 0.000,C 90.000,E1 54.895} C_DIS
LIN {X -0.211,Y -586.196,Z 1127.095,A 0.000,B 0.000,C 90.000,E1 53.050} C_DIS
LIN {X -0.267,Y -586.615,Z 1127.089,A 0.000,B 0.000,C 90.000,E1 51.984} C_DIS
LIN {X -0.223,Y -587.110,Z 1127.081,A 0.000,B 0.000,C 90.000,E1 50.642} C_DIS
LIN {X 0.092,Y -587.264,Z 1127.075,A 0.000,B 0.000,C 90.000,E1 49.542} C_DIS
LIN {X -0.045,Y -587.338,Z 1127.069,A 0.000,B 0.000,C 90.000,E1 48.485} C_DIS
LIN {X -0.042,Y -587.137,Z 1127.062,A 0.000,B 0.000,C 90.000,E1 47.148} C_DIS
LIN {X 0.213,Y -586.896,Z 1127.056,A 0.000,B 0.000,C 90.000,E1 46.053} C_DIS
LIN {X -0.210,Y -586.350,Z 1127.049,A 0.000,B 0.000,C 90.000,E1 44.757} C_DIS
LIN {X 0.034,Y -585.765,Z 1127.043,A 0.000,B 0.000,C 90.000,E1 43.662} C_DIS
LIN {X 0.099,Y -585.203,Z 1127.038,A 0.000,B 0.000,C 90.000,E1 42.852} C_DIS
LIN {X 0.235,Y -583.472,Z 1127.029,A 0.000,B 0.000,C 90.000,E1 41.229} C_DIS
LIN {X 0.048,Y -582.172,Z 1127.023,A 0.000,B 0.000,C 90.000,E1 40.172} C_DIS
LIN {X 0.119,Y -581.058,Z 1127.019,A 0.000,B 0.000,C 90.000,E1 39.358} C_DIS
LIN {X -0.108,Y -579.282,Z 1127.013,A 0.000,B 0.000,C 90.000,E1 38.302} C_DIS
LIN {X -0.264,Y -577.361,Z 1127.007,A 0.000,B 0.000,C 90.000,E1 37.237} C_DIS
LIN {X 0.211,Y -575.514,Z 1127.002,A 0.000,B 0.000,C 90.000,E1 36.377} C_DIS
LIN {X -0.140,Y -573.445,Z 1126.998,A 0.000,B 0.000,C 90.000,E1 35.598} C_DIS
LIN {X 0.147,Y -571.922,Z 1126.995,A 0.000,B 0.000,C 90.000,E1 35.025} C_DIS
LIN {X 0.354,Y -568.388,Z 1126.989,A 0.000,B 0.000,C 90.000,E1 33.913} C_DIS
LIN {X 0.086,Y -565.254,Z 1126.984,A 0.000,B 0.000,C 90.000,E1 33.118} C_DIS
LIN {X 0.100,Y -561.736,Z 1126.979,A 0.000,B 0.000,C 90.000,E1 32.291} C_DIS
LIN {X 0.175,Y -558.574,Z 1126.976,A 0.000,B 0.000,C 90.000,E1 31.592} C_DIS
LIN {X -0.189,Y -554.392,Z 1126.971,A 0.000,B 0.000,C 90.000,E1 30.797} C_DIS
LIN {X -0.075,Y -548.313,Z 1126.965,A 0.000,B 0.000,C 90.000,E1 29.667} C_DIS
LIN {X 0.063,Y -544.147,Z 1126.961,A 0.000,B 0.000,C 90.000,E1 28.949} C_DIS
LIN {X 0.291,Y -540.558,Z 1126.958,A 0.000,B 0.000,C 90.000,E1 28.359} C_DIS
LIN {X -0.123,Y -535.722,Z 1126.954,A 0.000,B 0.000,C 90.000,E1 27.692} C_DIS
LIN {X 0.127,Y -530.555,Z 1126.950,A 0.000,B 0.000,C 90.000,E1 26.950} C_DIS
LIN {X 0.095,Y -524.829,Z 1126.946,A 0.000,B 0.000,C 90.000,E1 26.232} C_DIS
LIN {X 0.312,Y -517.530,Z 1126.941,A 0.000,B 0.000,C 90.000,E1 25.335} C_DIS
LIN {X 0.130,Y -512.366,Z 1126.938,A 0.000,B 0.000,C 90.000,E1 24.771} C_DIS
LIN {X 0.170,Y -501.697,Z 1126.932,A 0.000,B 0.000,C 90.000,E1 23.643} C_DIS
LIN {X 0.018,Y -491.941,Z 1126.926,A 0.000,B 0.000,C 90.000,E1 22.695} C_DIS
LIN {X 0.252,Y -480.386,Z 1126.920,A 0.000,B 0.000,C 90.000,E1 21.589} C_DIS
LIN {X 0.082,Y -469.793,Z 1126.915,A 0.000,B 0.000,C 90.000,E1 20.684} C_DIS
LIN {X 0.105,Y -460.847,Z 1126.911,A 0.000,B 0.000,C 90.000,E1 19.885} C_DIS
LIN {X 0.009,Y -440.145,Z 1126.900,A 0.000,B 0.000,C 90.000,E1 18.000} C_DIS
LIN {X 0.147,Y -427.168,Z 1126.893,A 0.000,B 0.000,C 90.000,E1 16.677} C_DIS
LIN {X -0.153,Y -415.951,Z 1126.886,A 0.000,B 0.000,C 90.000,E1 15.481} C_DIS
LIN {X 0.061,Y -405.175,Z 1126.879,A 0.000,B 0.000,C 90.000,E1 14.120} C_DIS
LIN {X 0.155,Y -400.048,Z 1126.875,A 0.000,B 0.000,C 90.000,E1 13.411} C_DIS
LIN {X 0.179,Y -396.540,Z 1126.871,A 0.000,B 0.000,C 90.000,E1 12.827} C_DIS
LIN {X 0.177,Y -394.074,Z 1126.869,A 0.000,B 0.000,C 90.000,E1 12.299} C_DIS
LIN {X 0.202,Y -393.414,Z 1126.868,A 0.000,B 0.000,C 90.000,E1 12.119} C_DIS
LIN {X -0.030,Y -392.393,Z 1126.865,A 0.000,B 0.000,C 90.000,E1 11.771} C_DIS
LIN {X -0.044,Y -392.078,Z 1126.862,A 0.000,B 0.000,C 90.000,E1 11.243} C_DIS
LIN {X -0.070,Y -392.398,Z 1126.860,A 0.000,B 0.000,C 90.000,E1 10.894} C_DIS
LIN {X -0.114,Y -392.784,Z 1126.859,A 0.000,B 0.000,C 90.000,E1 10.546} C_DIS
LIN {X -0.200,Y -394.024,Z 1126.855,A 0.000,B 0.000,C 90.000,E1 9.849} C_DIS
LIN {X 0.080,Y -396.620,Z 1126.849,A 0.000,B 0.000,C 90.000,E1 8.746} C_DIS
LIN {X -0.112,Y -403.636,Z 1126.835,A 0.000,B 0.000,C 90.000,E1 6.315} C_DIS
LIN {X -0.143,Y -405.444,Z 1126.832,A 0.000,B 0.000,C 90.000,E1 5.796} C_DIS
LIN {X -0.145,Y -407.011,Z 1126.830,A 0.000,B 0.000,C 90.000,E1 5.448} C_DIS
LIN {X -0.163,Y -407.984,Z 1126.829,A 0.000,B 0.000,C 90.000,E1 5.277} C_DIS
LIN {X -0.160,Y -411.810,Z 1126.826,A 0.000,B 0.000,C 90.000,E1 4.759} C_DIS
LIN {X 0.149,Y -417.654,Z 1126.824,A 0.000,B 0.000,C 90.000,E1 4.245} C_DIS
LIN {X 0.064,Y -434.102,Z 1126.817,A 0.000,B 0.000,C 90.000,E1 3.094} C_DIS
LIN {X 0.087,Y -458.672,Z 1126.808,A 0.000,B 0.000,C 90.000,E1 1.432} C_DIS
LIN {X 0.118,Y -470.051,Z 1126.804,A 0.000,B 0.000,C 90.000,E1 0.688} C_DIS
LIN {X 0.008,Y -478.177,Z 1126.801,A 0.000,B 0.000,C 90.000,E1 0.172} C_DIS
LIN {X -0.172,Y -486.893,Z 1126.798,A 0.000,B 0.000,C 90.000,E1 359.599} C_DIS
LIN {X -0.052,Y -491.539,Z 1126.796,A 0.000,B 0.000,C 90.000,E1 359.255} C_DIS
LIN {X -0.009,Y -497.640,Z 1126.793,A 0.000,B 0.000,C 90.000,E1 358.797} C_DIS
LIN {X -0.070,Y -503.626,Z 1126.791,A 0.000,B 0.000,C 90.000,E1 358.339} C_DIS
LIN {X 0.215,Y -511.999,Z 1126.787,A 0.000,B 0.000,C 90.000,E1 357.593} C_DIS
LIN {X -0.119,Y -516.273,Z 1126.785,A 0.000,B 0.000,C 90.000,E1 357.249} C_DIS
LIN {X -0.066,Y -521.441,Z 1126.782,A 0.000,B 0.000,C 90.000,E1 356.731} C_DIS
LIN {X 0.127,Y -526.724,Z 1126.779,A 0.000,B 0.000,C 90.000,E1 356.159} C_DIS
LIN {X 0.173,Y -531.792,Z 1126.776,A 0.000,B 0.000,C 90.000,E1 355.584} C_DIS
LIN {X -0.086,Y -537.395,Z 1126.772,A 0.000,B 0.000,C 90.000,E1 354.894} C_DIS
LIN {X 0.233,Y -542.543,Z 1126.768,A 0.000,B 0.000,C 90.000,E1 354.147} C_DIS
LIN {X 0.119,Y -547.049,Z 1126.764,A 0.000,B 0.000,C 90.000,E1 353.451} C_DIS
LIN {X -0.018,Y -551.209,Z 1126.760,A 0.000,B 0.000,C 90.000,E1 352.761} C_DIS
LIN {X 0.128,Y -554.216,Z 1126.757,A 0.000,B 0.000,C 90.000,E1 352.186} C_DIS
LIN {X -0.177,Y -557.018,Z 1126.754,A 0.000,B 0.000,C 90.000,E1 351.659} C_DIS
LIN {X 0.008,Y -559.524,Z 1126.750,A 0.000,B 0.000,C 90.000,E1 351.084} C_DIS
LIN {X -0.200,Y -562.921,Z 1126.746,A 0.000,B 0.000,C 90.000,E1 350.274} C_DIS
LIN {X 0.277,Y -566.025,Z 1126.741,A 0.000,B 0.000,C 90.000,E1 349.398} C_DIS
LIN {X 0.238,Y -568.963,Z 1126.737,A 0.000,B 0.000,C 90.000,E1 348.578} C_DIS
LIN {X -0.137,Y -572.480,Z 1126.731,A 0.000,B 0.000,C 90.000,E1 347.521} C_DIS
LIN {X -0.107,Y -574.979,Z 1126.726,A 0.000,B 0.000,C 90.000,E1 346.700} C_DIS
LIN {X 0.152,Y -578.106,Z 1126.720,A 0.000,B 0.000,C 90.000,E1 345.589} C_DIS
LIN {X -0.150,Y -581.776,Z 1126.713,A 0.000,B 0.000,C 90.000,E1 344.267} C_DIS
LIN {X -0.211,Y -584.610,Z 1126.707,A 0.000,B 0.000,C 90.000,E1 343.196} C_DIS
LIN {X -0.241,Y -587.310,Z 1126.701,A 0.000,B 0.000,C 90.000,E1 342.127} C_DIS
LIN {X -0.060,Y -589.818,Z 1126.695,A 0.000,B 0.000,C 90.000,E1 341.040} C_DIS
LIN {X 0.153,Y -592.167,Z 1126.689,A 0.000,B 0.000,C 90.000,E1 339.953} C_DIS
LIN {X 0.177,Y -595.276,Z 1126.680,A 0.000,B 0.000,C 90.000,E1 338.358} C_DIS
LIN {X -0.020,Y -596.201,Z 1126.677,A 0.000,B 0.000,C 90.000,E1 337.847} C_DIS
LIN {X 0.028,Y -597.283,Z 1126.673,A 0.000,B 0.000,C 90.000,E1 337.050} C_DIS
LIN {X -0.005,Y -598.573,Z 1126.667,A 0.000,B 0.000,C 90.000,E1 335.997} C_DIS
LIN {X -0.245,Y -599.311,Z 1126.662,A 0.000,B 0.000,C 90.000,E1 335.229} C_DIS
LIN {X 0.070,Y -599.816,Z 1126.658,A 0.000,B 0.000,C 90.000,E1 334.409} C_DIS
LIN {X -0.151,Y -600.080,Z 1126.654,A 0.000,B 0.000,C 90.000,E1 333.640} C_DIS
LIN {X 0.166,Y -600.088,Z 1126.649,A 0.000,B 0.000,C 90.000,E1 332.820} C_DIS
LIN {X 0.225,Y -599.842,Z 1126.645,A 0.000,B 0.000,C 90.000,E1 332.025} C_DIS
LIN {X 0.076,Y -599.500,Z 1126.642,A 0.000,B 0.000,C 90.000,E1 331.513} C_DIS
LIN {X -0.076,Y -598.983,Z 1126.639,A 0.000,B 0.000,C 90.000,E1 331.001} C_DIS
LIN {X 0.193,Y -597.427,Z 1126.633,A 0.000,B 0.000,C 90.000,E1 329.921} C_DIS
LIN {X 0.235,Y -595.771,Z 1126.629,A 0.000,B 0.000,C 90.000,E1 329.125} C_DIS
LIN {X 0.259,Y -593.768,Z 1126.624,A 0.000,B 0.000,C 90.000,E1 328.329} C_DIS
LIN {X 0.157,Y -592.965,Z 1126.623,A 0.000,B 0.000,C 90.000,E1 328.074} C_DIS
LIN {X -0.038,Y -590.141,Z 1126.618,A 0.000,B 0.000,C 90.000,E1 327.296} C_DIS
LIN {X -0.079,Y -586.960,Z 1126.614,A 0.000,B 0.000,C 90.000,E1 326.501} C_DIS
LIN {X -0.023,Y -584.592,Z 1126.611,A 0.000,B 0.000,C 90.000,E1 325.960} C_DIS
LIN {X -0.293,Y -580.576,Z 1126.606,A 0.000,B 0.000,C 90.000,E1 325.182} C_DIS
LIN {X 0.045,Y -577.607,Z 1126.604,A 0.000,B 0.000,C 90.000,E1 324.609} C_DIS
LIN {X -0.333,Y -573.781,Z 1126.600,A 0.000,B 0.000,C 90.000,E1 323.989} C_DIS
LIN {X -0.043,Y -570.385,Z 1126.597,A 0.000,B 0.000,C 90.000,E1 323.417} C_DIS
LIN {X 0.109,Y -565.805,Z 1126.593,A 0.000,B 0.000,C 90.000,E1 322.718} C_DIS
LIN {X 0.213,Y -558.751,Z 1126.588,A 0.000,B 0.000,C 90.000,E1 321.743} C_DIS
LIN {X -0.030,Y -553.405,Z 1126.584,A 0.000,B 0.000,C 90.000,E1 321.090} C_DIS
LIN {X 0.245,Y -550.194,Z 1126.582,A 0.000,B 0.000,C 90.000,E1 320.642} C_DIS
LIN {X 0.024,Y -538.780,Z 1126.574,A 0.000,B 0.000,C 90.000,E1 319.256} C_DIS
LIN {X -0.014,Y -534.931,Z 1126.571,A 0.000,B 0.000,C 90.000,E1 318.690} C_DIS
LIN {X -0.017,Y -533.265,Z 1126.569,A 0.000,B 0.000,C 90.000,E1 318.405} C_DIS
LIN {X 0.156,Y -532.581,Z 1126.568,A 0.000,B 0.000,C 90.000,E1 318.243} C_DIS
LIN {X -0.126,Y -531.860,Z 1126.567,A 0.000,B 0.000,C 90.000,E1 318.081} C_DIS
LIN {X -0.144,Y -530.406,Z 1126.566,A 0.000,B 0.000,C 90.000,E1 317.796} C_DIS
LIN {X -0.232,Y -528.356,Z 1126.562,A 0.000,B 0.000,C 90.000,E1 317.229} C_DIS
LIN {X 0.055,Y -527.335,Z 1126.559,A 0.000,B 0.000,C 90.000,E1 316.620} C_DIS
LIN {X 0.215,Y -526.976,Z 1126.558,A 0.000,B 0.000,C 90.000,E1 316.458} C_DIS
LIN {X 0.019,Y -526.019,Z 1126.553,A 0.000,B 0.000,C 90.000,E1 315.567} C_DIS
LIN {X 0.110,Y -525.223,Z 1126.545,A 0.000,B 0.000,C 90.000,E1 314.109} C_DIS
LIN {X 0.075,Y -525.129,Z 1126.534,A 0.000,B 0.000,C 90.000,E1 312.081} C_DIS
LIN {X -0.109,Y -526.498,Z 1126.516,A 0.000,B 0.000,C 90.000,E1 308.910} C_DIS
LIN {X 0.044,Y -527.515,Z 1126.506,A 0.000,B 0.000,C 90.000,E1 307.156} C_DIS
LIN {X -0.106,Y -528.671,Z 1126.497,A 0.000,B 0.000,C 90.000,E1 305.438} C_DIS
LIN {X -0.087,Y -529.759,Z 1126.489,A 0.000,B 0.000,C 90.000,E1 303.992} C_DIS
LIN {X 0.076,Y -531.266,Z 1126.478,A 0.000,B 0.000,C 90.000,E1 301.957} C_DIS
LIN {X 0.005,Y -532.815,Z 1126.466,A 0.000,B 0.000,C 90.000,E1 299.951} C_DIS
LIN {X -0.165,Y -533.669,Z 1126.460,A 0.000,B 0.000,C 90.000,E1 298.821} C_DIS
LIN {X -0.147,Y -534.529,Z 1126.452,A 0.000,B 0.000,C 90.000,E1 297.385} C_DIS
LIN {X -0.081,Y -534.983,Z 1126.446,A 0.000,B 0.000,C 90.000,E1 296.232} C_DIS
LIN {X 0.270,Y -535.203,Z 1126.441,A 0.000,B 0.000,C 90.000,E1 295.335} C_DIS
LIN {X -0.167,Y -535.356,Z 1126.433,A 0.000,B 0.000,C 90.000,E1 293.951} C_DIS
LIN {X 0.303,Y -535.409,Z 1126.422,A 0.000,B 0.000,C 90.000,E1 291.897} C_DIS
LIN {X 0.153,Y -535.363,Z 1126.414,A 0.000,B 0.000,C 90.000,E1 290.482} C_DIS
LIN {X 0.020,Y -535.103,Z 1126.404,A 0.000,B 0.000,C 90.000,E1 288.779} C_DIS
LIN {X 0.183,Y -534.754,Z 1126.396,A 0.000,B 0.000,C 90.000,E1 287.330} C_DIS
LIN {X -0.012,Y -534.388,Z 1126.390,A 0.000,B 0.000,C 90.000,E1 286.205} C_DIS
LIN {X 0.028,Y -533.630,Z 1126.380,A 0.000,B 0.000,C 90.000,E1 284.481} C_DIS
LIN {X -0.130,Y -532.893,Z 1126.373,A 0.000,B 0.000,C 90.000,E1 283.063} C_DIS
LIN {X 0.253,Y -532.022,Z 1126.363,A 0.000,B 0.000,C 90.000,E1 281.299} C_DIS
LIN {X -0.117,Y -531.108,Z 1126.353,A 0.000,B 0.000,C 90.000,E1 279.613} C_DIS
LIN {X 0.017,Y -530.183,Z 1126.344,A 0.000,B 0.000,C 90.000,E1 277.871} C_DIS
LIN {X -0.020,Y -529.065,Z 1126.331,A 0.000,B 0.000,C 90.000,E1 275.568} C_DIS
LIN {X -0.067,Y -528.326,Z 1126.321,A 0.000,B 0.000,C 90.000,E1 273.841} C_DIS
LIN {X -0.210,Y -527.409,Z 1126.310,A 0.000,B 0.000,C 90.000,E1 271.833} C_DIS
LIN {X 0.180,Y -526.747,Z 1126.302,A 0.000,B 0.000,C 90.000,E1 270.344} C_DIS
LIN {X 0.002,Y -525.968,Z 1126.292,A 0.000,B 0.000,C 90.000,E1 268.625} C_DIS
LIN {X -0.149,Y -525.285,Z 1126.284,A 0.000,B 0.000,C 90.000,E1 267.192} C_DIS
LIN {X -0.234,Y -524.744,Z 1126.280,A 0.000,B 0.000,C 90.000,E1 266.331} C_DIS
LIN {X 0.149,Y -523.700,Z 1126.270,A 0.000,B 0.000,C 90.000,E1 264.546} C_DIS
LIN {X 0.044,Y -522.997,Z 1126.265,A 0.000,B 0.000,C 90.000,E1 263.685} C_DIS
LIN {X -0.078,Y -521.561,Z 1126.257,A 0.000,B 0.000,C 90.000,E1 262.243} C_DIS
LIN {X -0.154,Y -519.658,Z 1126.246,A 0.000,B 0.000,C 90.000,E1 260.208} C_DIS
LIN {X -0.272,Y -517.959,Z 1126.236,A 0.000,B 0.000,C 90.000,E1 258.465} C_DIS
LIN {X -0.256,Y -515.686,Z 1126.223,A 0.000,B 0.000,C 90.000,E1 256.117} C_DIS
LIN {X -0.135,Y -514.039,Z 1126.213,A 0.000,B 0.000,C 90.000,E1 254.338} C_DIS
LIN {X 0.201,Y -511.964,Z 1126.202,A 0.000,B 0.000,C 90.000,E1 252.236} C_DIS
LIN {X -0.053,Y -510.437,Z 1126.193,A 0.000,B 0.000,C 90.000,E1 250.786} C_DIS
LIN {X -0.239,Y -508.413,Z 1126.183,A 0.000,B 0.000,C 90.000,E1 249.028} C_DIS
LIN {X -0.207,Y -506.728,Z 1126.175,A 0.000,B 0.000,C 90.000,E1 247.539} C_DIS
LIN {X -0.205,Y -504.793,Z 1126.167,A 0.000,B 0.000,C 90.000,E1 246.049} C_DIS
LIN {X -0.117,Y -503.156,Z 1126.160,A 0.000,B 0.000,C 90.000,E1 244.845} C_DIS
LIN {X -0.079,Y -500.167,Z 1126.149,A 0.000,B 0.000,C 90.000,E1 242.743} C_DIS
LIN {X 0.052,Y -497.319,Z 1126.139,A 0.000,B 0.000,C 90.000,E1 240.923} C_DIS
LIN {X -0.069,Y -494.380,Z 1126.128,A 0.000,B 0.000,C 90.000,E1 239.125} C_DIS
LIN {X 0.007,Y -491.322,Z 1126.118,A 0.000,B 0.000,C 90.000,E1 237.296} C_DIS
LIN {X -0.074,Y -489.272,Z 1126.112,A 0.000,B 0.000,C 90.000,E1 236.087} C_DIS
LIN {X -0.260,Y -486.073,Z 1126.101,A 0.000,B 0.000,C 90.000,E1 234.276} C_DIS
LIN {X 0.118,Y -483.967,Z 1126.095,A 0.000,B 0.000,C 90.000,E1 233.004} C_DIS
LIN {X 0.074,Y -481.782,Z 1126.088,A 0.000,B 0.000,C 90.000,E1 231.778} C_DIS
LIN {X 0.209,Y -478.376,Z 1126.078,A 0.000,B 0.000,C 90.000,E1 229.908} C_DIS
LIN {X -0.088,Y -474.976,Z 1126.067,A 0.000,B 0.000,C 90.000,E1 228.081} C_DIS
LIN {X -0.145,Y -471.550,Z 1126.057,A 0.000,B 0.000,C 90.000,E1 226.215} C_DIS
LIN {X -0.138,Y -467.299,Z 1126.043,A 0.000,B 0.000,C 90.000,E1 223.704} C_DIS
LIN {X 0.290,Y -464.372,Z 1126.032,A 0.000,B 0.000,C 90.000,E1 221.757} C_DIS
LIN {X 0.040,Y -461.618,Z 1126.022,A 0.000,B 0.000,C 90.000,E1 219.886} C_DIS
LIN {X -0.048,Y -457.912,Z 1126.006,A 0.000,B 0.000,C 90.000,E1 217.030} C_DIS
LIN {X -0.103,Y -456.080,Z 1125.997,A 0.000,B 0.000,C 90.000,E1 215.438} C_DIS
LIN {X 0.001,Y -453.880,Z 1125.986,A 0.000,B 0.000,C 90.000,E1 213.499} C_DIS
LIN {X 0.077,Y -451.213,Z 1125.970,A 0.000,B 0.000,C 90.000,E1 210.590} C_DIS
LIN {X -0.195,Y -450.279,Z 1125.963,A 0.000,B 0.000,C 90.000,E1 209.333} C_DIS
LIN {X -0.147,Y -449.344,Z 1125.952,A 0.000,B 0.000,C 90.000,E1 207.385} C_DIS
LIN {X 0.143,Y -449.155,Z 1125.945,A 0.000,B 0.000,C 90.000,E1 206.052} C_DIS
LIN {X -0.096,Y -449.702,Z 1125.936,A 0.000,B 0.000,C 90.000,E1 204.463} C_DIS
LIN {X 0.138,Y -450.508,Z 1125.931,A 0.000,B 0.000,C 90.000,E1 203.462} C_DIS
LIN {X -0.037,Y -451.810,Z 1125.925,A 0.000,B 0.000,C 90.000,E1 202.514} C_DIS
LIN {X -0.060,Y -454.038,Z 1125.918,A 0.000,B 0.000,C 90.000,E1 201.227} C_DIS
LIN {X 0.193,Y -458.423,Z 1125.907,A 0.000,B 0.000,C 90.000,E1 199.268} C_DIS
LIN {X 0.185,Y -465.057,Z 1125.895,A 0.000,B 0.000,C 90.000,E1 197.040} C_DIS
LIN {X 0.045,Y -473.694,Z 1125.881,A 0.000,B 0.000,C 90.000,E1 194.537} C_DIS
LIN {X 0.016,Y -484.908,Z 1125.865,A 0.000,B 0.000,C 90.000,E1 191.591} C_DIS
LIN {X -0.079,Y -492.942,Z 1125.853,A 0.000,B 0.000,C 90.000,E1 189.613} C_DIS
LIN {X -0.050,Y -501.042,Z 1125.843,A 0.000,B 0.000,C 90.000,E1 187.644} C_DIS
LIN {X -0.217,Y -506.557,Z 1125.835,A 0.000,B 0.000,C 90.000,E1 186.315} C_DIS
LIN {X 0.160,Y -511.979,Z 1125.828,A 0.000,B 0.000,C 90.000,E1 184.935} C_DIS
LIN {X 0.197,Y -516.252,Z 1125.822,A 0.000,B 0.000,C 90.000,E1 183.898} C_DIS
LIN {X 0.097,Y -524.197,Z 1125.811,A 0.000,B 0.000,C 90.000,E1 182.007} C_DIS
LIN {X -0.083,Y -532.655,Z 1125.800,A 0.000,B 0.000,C 90.000,E1 180.000} C_DIS
LIN {X -0.098,Y -537.535,Z 1125.794,A 0.000,B 0.000,C 90.000,E1 178.854} C_DIS
LIN {X -0.265,Y -544.175,Z 1125.785,A 0.000,B 0.000,C 90.000,E1 177.306} C_DIS
LIN {X 0.030,Y -551.443,Z 1125.776,A 0.000,B 0.000,C 90.000,E1 175.584} C_DIS
LIN {X 0.051,Y -559.910,Z 1125.765,A 0.000,B 0.000,C 90.000,E1 173.628} C_DIS
LIN {X 0.252,Y -567.172,Z 1125.755,A 0.000,B 0.000,C 90.000,E1 171.951} C_DIS
LIN {X 0.042,Y -574.294,Z 1125.746,A 0.000,B 0.000,C 90.000,E1 170.330} C_DIS
LIN {X 0.301,Y -578.951,Z 1125.740,A 0.000,B 0.000,C 90.000,E1 169.218} C_DIS
LIN {X 0.180,Y -584.469,Z 1125.733,A 0.000,B 0.000,C 90.000,E1 167.881} C_DIS
LIN {X -0.053,Y -590.950,Z 1125.724,A 0.000,B 0.000,C 90.000,E1 166.297} C_DIS
LIN {X 0.007,Y -595.062,Z 1125.718,A 0.000,B 0.000,C 90.000,E1 165.227} C_DIS
LIN {X -0.153,Y -597.964,Z 1125.714,A 0.000,B 0.000,C 90.000,E1 164.448} C_DIS
LIN {X 0.013,Y -601.626,Z 1125.708,A 0.000,B 0.000,C 90.000,E1 163.378} C_DIS
LIN {X 0.134,Y -605.908,Z 1125.700,A 0.000,B 0.000,C 90.000,E1 162.054} C_DIS
LIN {X -0.250,Y -609.993,Z 1125.693,A 0.000,B 0.000,C 90.000,E1 160.786} C_DIS
LIN {X 0.212,Y -613.803,Z 1125.686,A 0.000,B 0.000,C 90.000,E1 159.444} C_DIS
LIN {X -0.093,Y -618.067,Z 1125.677,A 0.000,B 0.000,C 90.000,E1 157.922} C_DIS
LIN {X 0.155,Y -621.454,Z 1125.670,A 0.000,B 0.000,C 90.000,E1 156.613} C_DIS
LIN {X -0.107,Y -624.702,Z 1125.663,A 0.000,B 0.000,C 90.000,E1 155.357} C_DIS
LIN {X -0.047,Y -627.844,Z 1125.656,A 0.000,B 0.000,C 90.000,E1 154.076} C_DIS
LIN {X 0.073,Y -630.866,Z 1125.649,A 0.000,B 0.000,C 90.000,E1 152.794} C_DIS
LIN {X 0.167,Y -632.560,Z 1125.645,A 0.000,B 0.000,C 90.000,E1 152.025} C_DIS
LIN {X -0.164,Y -635.854,Z 1125.636,A 0.000,B 0.000,C 90.000,E1 150.539} C_DIS
LIN {X -0.180,Y -638.491,Z 1125.629,A 0.000,B 0.000,C 90.000,E1 149.282} C_DIS
LIN {X 0.130,Y -640.517,Z 1125.624,A 0.000,B 0.000,C 90.000,E1 148.250} C_DIS
LIN {X 0.051,Y -643.360,Z 1125.615,A 0.000,B 0.000,C 90.000,E1 146.755} C_DIS
LIN {X 0.079,Y -645.193,Z 1125.610,A 0.000,B 0.000,C 90.000,E1 145.754} C_DIS
LIN {X -0.146,Y -647.321,Z 1125.603,A 0.000,B 0.000,C 90.000,E1 144.529} C_DIS
LIN {X -0.187,Y -649.435,Z 1125.596,A 0.000,B 0.000,C 90.000,E1 143.290} C_DIS
LIN {X 0.037,Y -652.423,Z 1125.586,A 0.000,B 0.000,C 90.000,E1 141.537} C_DIS
LIN {X 0.351,Y -654.700,Z 1125.579,A 0.000,B 0.000,C 90.000,E1 140.275} C_DIS
LIN {X -0.265,Y -657.451,Z 1125.571,A 0.000,B 0.000,C 90.000,E1 138.852} C_DIS
LIN {X -0.400,Y -660.340,Z 1125.563,A 0.000,B 0.000,C 90.000,E1 137.391} C_DIS
LIN {X -0.058,Y -664.841,Z 1125.551,A 0.000,B 0.000,C 90.000,E1 135.162} C_DIS
LIN {X -0.061,Y -669.862,Z 1125.539,A 0.000,B 0.000,C 90.000,E1 132.975} C_DIS
LIN {X 0.059,Y -673.933,Z 1125.529,A 0.000,B 0.000,C 90.000,E1 131.272} C_DIS
LIN {X -0.220,Y -676.817,Z 1125.523,A 0.000,B 0.000,C 90.000,E1 130.092} C_DIS
LIN {X -0.233,Y -682.355,Z 1125.511,A 0.000,B 0.000,C 90.000,E1 127.935} C_DIS
LIN {X -0.029,Y -684.200,Z 1125.507,A 0.000,B 0.000,C 90.000,E1 127.202} C_DIS
LIN {X -0.387,Y -687.745,Z 1125.499,A 0.000,B 0.000,C 90.000,E1 125.804} C_DIS
LIN {X 0.292,Y -691.244,Z 1125.491,A 0.000,B 0.000,C 90.000,E1 124.326} C_DIS
LIN {X -0.184,Y -693.577,Z 1125.486,A 0.000,B 0.000,C 90.000,E1 123.420} C_DIS
LIN {X -0.054,Y -695.815,Z 1125.480,A 0.000,B 0.000,C 90.000,E1 122.467} C_DIS
LIN {X 0.353,Y -698.383,Z 1125.474,A 0.000,B 0.000,C 90.000,E1 121.258} C_DIS
LIN {X 0.184,Y -700.085,Z 1125.469,A 0.000,B 0.000,C 90.000,E1 120.335} C_DIS
LIN {X 0.251,Y -702.891,Z 1125.460,A 0.000,B 0.000,C 90.000,E1 118.693} C_DIS
LIN {X -0.147,Y -704.032,Z 1125.456,A 0.000,B 0.000,C 90.000,E1 118.025} C_DIS
LIN {X 0.081,Y -704.864,Z 1125.452,A 0.000,B 0.000,C 90.000,E1 117.308} C_DIS
LIN {X -0.003,Y -705.442,Z 1125.448,A 0.000,B 0.000,C 90.000,E1 116.616} C_DIS
LIN {X 0.220,Y -706.063,Z 1125.443,A 0.000,B 0.000,C 90.000,E1 115.668} C_DIS
LIN {X 0.166,Y -706.291,Z 1125.440,A 0.000,B 0.000,C 90.000,E1 115.207} C_DIS
LIN {X 0.103,Y -706.040,Z 1125.436,A 0.000,B 0.000,C 90.000,E1 114.515} C_DIS
LIN {X -0.250,Y -705.225,Z 1125.434,A 0.000,B 0.000,C 90.000,E1 114.079} C_DIS
LIN {X 0.038,Y -704.570,Z 1125.432,A 0.000,B 0.000,C 90.000,E1 113.823} C_DIS
LIN {X -0.322,Y -702.649,Z 1125.430,A 0.000,B 0.000,C 90.000,E1 113.387} C_DIS
LIN {X -0.182,Y -701.963,Z 1125.429,A 0.000,B 0.000,C 90.000,E1 113.259} C_DIS
LIN {X 0.086,Y -697.690,Z 1125.427,A 0.000,B 0.000,C 90.000,E1 112.770} C_DIS
LIN {X 0.218,Y -696.441,Z 1125.426,A 0.000,B 0.000,C 90.000,E1 112.642} C_DIS
LIN {X 0.384,Y -694.548,Z 1125.425,A 0.000,B 0.000,C 90.000,E1 112.514} C_DIS
LIN {X -0.153,Y -686.358,Z 1125.424,A 0.000,B 0.000,C 90.000,E1 112.259} C_DIS
LIN {X -0.255,Y -683.067,Z 1125.423,A 0.000,B 0.000,C 90.000,E1 112.206} C_DIS
LIN {X 0.205,Y -676.244,Z 1125.423,A 0.000,B 0.000,C 90.000,E1 112.099} C_DIS
LIN {X 0.136,Y -603.207,Z 1125.423,A 0.000,B 0.000,C 90.000,E1 112.099} C_DIS
LIN {X -0.064,Y -599.729,Z 1125.422,A 0.000,B 0.000,C 90.000,E1 111.897} C_DIS
LIN {X 0.078,Y -595.247,Z 1125.420,A 0.000,B 0.000,C 90.000,E1 111.535} C_DIS
LIN {X -0.153,Y -579.638,Z 1125.412,A 0.000,B 0.000,C 90.000,E1 110.174} C_DIS
LIN {X -0.041,Y -573.949,Z 1125.409,A 0.000,B 0.000,C 90.000,E1 109.685} C_DIS
LIN {X 0.143,Y -567.942,Z 1125.407,A 0.000,B 0.000,C 90.000,E1 109.214} C_DIS
LIN {X -0.188,Y -561.532,Z 1125.405,A 0.000,B 0.000,C 90.000,E1 108.833} C_DIS
LIN {X 0.107,Y -554.830,Z 1125.402,A 0.000,B 0.000,C 90.000,E1 108.417} C_DIS
LIN {X -0.203,Y -550.387,Z 1125.401,A 0.000,B 0.000,C 90.000,E1 108.127} C_DIS
LIN {X -0.257,Y -549.286,Z 1125.400,A 0.000,B 0.000,C 90.000,E1 107.946} C_DIS
LIN {X -0.129,Y -549.275,Z 1125.400,A 0.000,B 0.000,C 90.000,E1 107.928} C_DIS
LIN {X 0.190,Y -548.987,Z 1125.398,A 0.000,B 0.000,C 90.000,E1 107.583} C_DIS
LIN {X 0.064,Y -550.360,Z 1125.385,A 0.000,B 0.000,C 90.000,E1 105.300} C_DIS
LIN {X -0.103,Y -551.881,Z 1125.374,A 0.000,B 0.000,C 90.000,E1 103.355} C_DIS
LIN {X -0.225,Y -553.831,Z 1125.362,A 0.000,B 0.000,C 90.000,E1 101.130} C_DIS
LIN {X 0.023,Y -555.618,Z 1125.351,A 0.000,B 0.000,C 90.000,E1 99.151} C_DIS
LIN {X 0.226,Y -557.452,Z 1125.340,A 0.000,B 0.000,C 90.000,E1 97.182} C_DIS
LIN {X -0.286,Y -559.040,Z 1125.331,A 0.000,B 0.000,C 90.000,E1 95.568} C_DIS
LIN {X 0.216,Y -560.237,Z 1125.323,A 0.000,B 0.000,C 90.000,E1 94.131} C_DIS
LIN {X 0.175,Y -561.291,Z 1125.315,A 0.000,B 0.000,C 90.000,E1 92.751} C_DIS
LIN {X 0.116,Y -562.217,Z 1125.308,A 0.000,B 0.000,C 90.000,E1 91.375} C_DIS
LIN {X 0.268,Y -563.394,Z 1125.297,A 0.000,B 0.000,C 90.000,E1 89.427} C_DIS
LIN {X -0.102,Y -564.468,Z 1125.286,A 0.000,B 0.000,C 90.000,E1 87.535} C_DIS
LIN {X 0.142,Y -565.410,Z 1125.276,A 0.000,B 0.000,C 90.000,E1 85.584} C_DIS
LIN {X -0.212,Y -566.116,Z 1125.266,A 0.000,B 0.000,C 90.000,E1 83.970} C_DIS
LIN {X 0.179,Y -566.952,Z 1125.256,A 0.000,B 0.000,C 90.000,E1 82.008} C_DIS
LIN {X 0.100,Y -567.728,Z 1125.245,A 0.000,B 0.000,C 90.000,E1 80.095} C_DIS
LIN {X -0.247,Y -568.687,Z 1125.233,A 0.000,B 0.000,C 90.000,E1 77.937} C_DIS
LIN {X 0.101,Y -569.321,Z 1125.225,A 0.000,B 0.000,C 90.000,E1 76.533} C_DIS
LIN {X 0.175,Y -570.477,Z 1125.213,A 0.000,B 0.000,C 90.000,E1 74.338} C_DIS
LIN {X 0.292,Y -571.352,Z 1125.206,A 0.000,B 0.000,C 90.000,E1 72.960} C_DIS
LIN {X 0.053,Y -572.563,Z 1125.196,A 0.000,B 0.000,C 90.000,E1 71.348} C_DIS
LIN {X 0.191,Y -574.415,Z 1125.184,A 0.000,B 0.000,C 90.000,E1 69.156} C_DIS
LIN {X -0.099,Y -576.156,Z 1125.174,A 0.000,B 0.000,C 90.000,E1 67.283} C_DIS
LIN {X -0.260,Y -576.935,Z 1125.169,A 0.000,B 0.000,C 90.000,E1 66.485} C_DIS
LIN {X 0.277,Y -578.536,Z 1125.159,A 0.000,B 0.000,C 90.000,E1 64.537} C_DIS
LIN {X 0.081,Y -579.692,Z 1125.151,A 0.000,B 0.000,C 90.000,E1 63.204} C_DIS
LIN {X 0.026,Y -580.936,Z 1125.142,A 0.000,B 0.000,C 90.000,E1 61.591} C_DIS
LIN {X -0.232,Y -582.103,Z 1125.133,A 0.000,B 0.000,C 90.000,E1 59.999} C_DIS
LIN {X 0.199,Y -583.278,Z 1125.123,A 0.000,B 0.000,C 90.000,E1 58.074} C_DIS
LIN {X -0.022,Y -584.316,Z 1125.112,A 0.000,B 0.000,C 90.000,E1 56.215} C_DIS
LIN {X -0.066,Y -585.191,Z 1125.103,A 0.000,B 0.000,C 90.000,E1 54.609} C_DIS
LIN {X 0.087,Y -586.108,Z 1125.093,A 0.000,B 0.000,C 90.000,E1 52.718} C_DIS
LIN {X 0.194,Y -586.424,Z 1125.089,A 0.000,B 0.000,C 90.000,E1 51.904} C_DIS
LIN {X -0.134,Y -586.895,Z 1125.081,A 0.000,B 0.000,C 90.000,E1 50.598} C_DIS
LIN {X -0.090,Y -587.052,Z 1125.074,A 0.000,B 0.000,C 90.000,E1 49.256} C_DIS
LIN {X 0.157,Y -587.034,Z 1125.068,A 0.000,B 0.000,C 90.000,E1 48.162} C_DIS
LIN {X -0.091,Y -586.730,Z 1125.059,A 0.000,B 0.000,C 90.000,E1 46.581} C_DIS
LIN {X -0.093,Y -586.279,Z 1125.051,A 0.000,B 0.000,C 90.000,E1 45.243} C_DIS
LIN {X 0.302,Y -585.566,Z 1125.044,A 0.000,B 0.000,C 90.000,E1 43.866} C_DIS
LIN {X 0.274,Y -584.527,Z 1125.036,A 0.000,B 0.000,C 90.000,E1 42.528} C_DIS
LIN {X -0.166,Y -583.050,Z 1125.029,A 0.000,B 0.000,C 90.000,E1 41.229} C_DIS
LIN {X -0.086,Y -582.089,Z 1125.025,A 0.000,B 0.000,C 90.000,E1 40.415} C_DIS
LIN {X 0.077,Y -580.604,Z 1125.019,A 0.000,B 0.000,C 90.000,E1 39.322} C_DIS
LIN {X -0.235,Y -579.289,Z 1125.014,A 0.000,B 0.000,C 90.000,E1 38.543} C_DIS
LIN {X 0.124,Y -576.832,Z 1125.007,A 0.000,B 0.000,C 90.000,E1 37.156} C_DIS
LIN {X -0.214,Y -574.912,Z 1125.002,A 0.000,B 0.000,C 90.000,E1 36.377} C_DIS
LIN {X 0.231,Y -572.811,Z 1124.998,A 0.000,B 0.000,C 90.000,E1 35.518} C_DIS
LIN {X -0.285,Y -571.246,Z 1124.995,A 0.000,B 0.000,C 90.000,E1 35.025} C_DIS
LIN {X -0.086,Y -567.649,Z 1124.988,A 0.000,B 0.000,C 90.000,E1 33.913} C_DIS
LIN {X -0.050,Y -564.446,Z 1124.984,A 0.000,B 0.000,C 90.000,E1 33.086} C_DIS
LIN {X -0.155,Y -560.286,Z 1124.979,A 0.000,B 0.000,C 90.000,E1 32.133} C_DIS
LIN {X 0.266,Y -556.291,Z 1124.974,A 0.000,B 0.000,C 90.000,E1 31.258} C_DIS
LIN {X 0.107,Y -553.433,Z 1124.971,A 0.000,B 0.000,C 90.000,E1 30.718} C_DIS
LIN {X -0.070,Y -547.293,Z 1124.965,A 0.000,B 0.000,C 90.000,E1 29.617} C_DIS
LIN {X -0.291,Y -543.970,Z 1124.961,A 0.000,B 0.000,C 90.000,E1 29.077} C_DIS
LIN {X -0.062,Y -540.393,Z 1124.958,A 0.000,B 0.000,C 90.000,E1 28.487} C_DIS
LIN {X 0.137,Y -536.588,Z 1124.955,A 0.000,B 0.000,C 90.000,E1 27.897} C_DIS
LIN {X 0.059,Y -532.510,Z 1124.952,A 0.000,B 0.000,C 90.000,E1 27.334} C_DIS
LIN {X 0.197,Y -528.188,Z 1124.949,A 0.000,B 0.000,C 90.000,E1 26.744} C_DIS
LIN {X -0.087,Y -522.343,Z 1124.945,A 0.000,B 0.000,C 90.000,E1 26.052} C_DIS
LIN {X 0.108,Y -514.850,Z 1124.940,A 0.000,B 0.000,C 90.000,E1 25.155} C_DIS
LIN {X 0.138,Y -510.902,Z 1124.938,A 0.000,B 0.000,C 90.000,E1 24.719} C_DIS
LIN {X -0.116,Y -502.148,Z 1124.932,A 0.000,B 0.000,C 90.000,E1 23.823} C_DIS
LIN {X 0.272,Y -495.105,Z 1124.928,A 0.000,B 0.000,C 90.000,E1 23.078} C_DIS
LIN {X -0.153,Y -489.553,Z 1124.925,A 0.000,B 0.000,C 90.000,E1 22.589} C_DIS
LIN {X -0.097,Y -480.845,Z 1124.921,A 0.000,B 0.000,C 90.000,E1 21.770} C_DIS
LIN {X 0.157,Y -472.137,Z 1124.917,A 0.000,B 0.000,C 90.000,E1 20.972} C_DIS
LIN {X -0.204,Y -462.030,Z 1124.912,A 0.000,B 0.000,C 90.000,E1 20.120} C_DIS
LIN {X -0.062,Y -440.153,Z 1124.901,A 0.000,B 0.000,C 90.000,E1 18.109} C_DIS
LIN {X -0.117,Y -425.886,Z 1124.893,A 0.000,B 0.000,C 90.000,E1 16.677} C_DIS
LIN {X 0.193,Y -413.485,Z 1124.885,A 0.000,B 0.000,C 90.000,E1 15.245} C_DIS
LIN {X 0.139,Y -403.240,Z 1124.878,A 0.000,B 0.000,C 90.000,E1 13.953} C_DIS
LIN {X -0.027,Y -399.566,Z 1124.875,A 0.000,B 0.000,C 90.000,E1 13.467} C_DIS
LIN {X 0.022,Y -395.561,Z 1124.871,A 0.000,B 0.000,C 90.000,E1 12.771} C_DIS
LIN {X 0.019,Y -393.337,Z 1124.868,A 0.000,B 0.000,C 90.000,E1 12.243} C_DIS
LIN {X 0.061,Y -392.485,Z 1124.866,A 0.000,B 0.000,C 90.000,E1 11.883} C_DIS
LIN {X -0.137,Y -392.252,Z 1124.865,A 0.000,B 0.000,C 90.000,E1 11.771} C_DIS
LIN {X 0.082,Y -392.073,Z 1124.863,A 0.000,B 0.000,C 90.000,E1 11.243} C_DIS
LIN {X 0.037,Y -392.408,Z 1124.861,A 0.000,B 0.000,C 90.000,E1 10.894} C_DIS
LIN {X -0.052,Y -393.422,Z 1124.857,A 0.000,B 0.000,C 90.000,E1 10.197} C_DIS
LIN {X -0.132,Y -394.852,Z 1124.853,A 0.000,B 0.000,C 90.000,E1 9.500} C_DIS
LIN {X -0.010,Y -404.618,Z 1124.833,A 0.000,B 0.000,C 90.000,E1 5.967} C_DIS
LIN {X -0.073,Y -406.648,Z 1124.830,A 0.000,B 0.000,C 90.000,E1 5.454} C_DIS
LIN {X -0.053,Y -407.523,Z 1124.829,A 0.000,B 0.000,C 90.000,E1 5.277} C_DIS
LIN {X 0.129,Y -411.969,Z 1124.826,A 0.000,B 0.000,C 90.000,E1 4.645} C_DIS
LIN {X -0.210,Y -416.666,Z 1124.824,A 0.000,B 0.000,C 90.000,E1 4.302} C_DIS
LIN {X 0.171,Y -432.255,Z 1124.818,A 0.000,B 0.000,C 90.000,E1 3.154} C_DIS
LIN {X -0.118,Y -460.117,Z 1124.807,A 0.000,B 0.000,C 90.000,E1 1.318} C_DIS
LIN {X -0.017,Y -473.127,Z 1124.803,A 0.000,B 0.000,C 90.000,E1 0.458} C_DIS
LIN {X -0.219,Y -484.703,Z 1124.798,A 0.000,B 0.000,C 90.000,E1 359.714} C_DIS
LIN {X -0.007,Y -490.900,Z 1124.796,A 0.000,B 0.000,C 90.000,E1 359.255} C_DIS
LIN {X 0.193,Y -498.327,Z 1124.793,A 0.000,B 0.000,C 90.000,E1 358.682} C_DIS
LIN {X 0.116,Y -502.932,Z 1124.791,A 0.000,B 0.000,C 90.000,E1 358.339} C_DIS
LIN {X -0.185,Y -510.261,Z 1124.787,A 0.000,B 0.000,C 90.000,E1 357.764} C_DIS
LIN {X -0.221,Y -517.263,Z 1124.784,A 0.000,B 0.000,C 90.000,E1 357.135} C_DIS
LIN {X -0.100,Y -525.169,Z 1124.780,A 0.000,B 0.000,C 90.000,E1 356.331} C_DIS
LIN {X -0.241,Y -531.555,Z 1124.776,A 0.000,B 0.000,C 90.000,E1 355.641} C_DIS
LIN {X 0.051,Y -537.224,Z 1124.772,A 0.000,B 0.000,C 90.000,E1 354.894} C_DIS
LIN {X 0.098,Y -541.439,Z 1124.769,A 0.000,B 0.000,C 90.000,E1 354.318} C_DIS
LIN {X -0.088,Y -546.147,Z 1124.765,A 0.000,B 0.000,C 90.000,E1 353.628} C_DIS
LIN {X -0.170,Y -550.375,Z 1124.761,A 0.000,B 0.000,C 90.000,E1 352.932} C_DIS
LIN {X -0.029,Y -553.543,Z 1124.758,A 0.000,B 0.000,C 90.000,E1 352.356} C_DIS
LIN {X 0.133,Y -556.452,Z 1124.755,A 0.000,B 0.000,C 90.000,E1 351.781} C_DIS
LIN {X 0.147,Y -559.611,Z 1124.751,A 0.000,B 0.000,C 90.000,E1 351.084} C_DIS
LIN {X -0.116,Y -561.956,Z 1124.748,A 0.000,B 0.000,C 90.000,E1 350.557} C_DIS
LIN {X 0.255,Y -565.148,Z 1124.743,A 0.000,B 0.000,C 90.000,E1 349.690} C_DIS
LIN {X -0.175,Y -569.147,Z 1124.737,A 0.000,B 0.000,C 90.000,E1 348.634} C_DIS
LIN {X 0.207,Y -573.555,Z 1124.729,A 0.000,B 0.000,C 90.000,E1 347.229} C_DIS
LIN {X 0.247,Y -576.037,Z 1124.725,A 0.000,B 0.000,C 90.000,E1 346.408} C_DIS
LIN {X 0.321,Y -579.914,Z 1124.717,A 0.000,B 0.000,C 90.000,E1 345.046} C_DIS
LIN {X 0.122,Y -584.273,Z 1124.708,A 0.000,B 0.000,C 90.000,E1 343.449} C_DIS
LIN {X -0.068,Y -587.663,Z 1124.701,A 0.000,B 0.000,C 90.000,E1 342.127} C_DIS
LIN {X -0.012,Y -590.784,Z 1124.693,A 0.000,B 0.000,C 90.000,E1 340.786} C_DIS
LIN {X 0.221,Y -593.119,Z 1124.687,A 0.000,B 0.000,C 90.000,E1 339.699} C_DIS
LIN {X 0.272,Y -596.218,Z 1124.679,A 0.000,B 0.000,C 90.000,E1 338.103} C_DIS
LIN {X -0.234,Y -597.452,Z 1124.674,A 0.000,B 0.000,C 90.000,E1 337.358} C_DIS
LIN {X -0.344,Y -599.055,Z 1124.667,A 0.000,B 0.000,C 90.000,E1 336.049} C_DIS
LIN {X -0.032,Y -599.841,Z 1124.662,A 0.000,B 0.000,C 90.000,E1 335.229} C_DIS
LIN {X 0.289,Y -600.383,Z 1124.658,A 0.000,B 0.000,C 90.000,E1 334.409} C_DIS
LIN {X 0.074,Y -600.694,Z 1124.654,A 0.000,B 0.000,C 90.000,E1 333.640} C_DIS
LIN {X -0.136,Y -600.758,Z 1124.649,A 0.000,B 0.000,C 90.000,E1 332.871} C_DIS
LIN {X -0.348,Y -600.574,Z 1124.645,A 0.000,B 0.000,C 90.000,E1 332.103} C_DIS
LIN {X 0.247,Y -600.075,Z 1124.641,A 0.000,B 0.000,C 90.000,E1 331.257} C_DIS
LIN {X 0.312,Y -599.171,Z 1124.636,A 0.000,B 0.000,C 90.000,E1 330.461} C_DIS
LIN {X 0.153,Y -598.367,Z 1124.633,A 0.000,B 0.000,C 90.000,E1 329.950} C_DIS
LIN {X -0.094,Y -596.244,Z 1124.627,A 0.000,B 0.000,C 90.000,E1 328.918} C_DIS
LIN {X -0.065,Y -594.137,Z 1124.623,A 0.000,B 0.000,C 90.000,E1 328.122} C_DIS
LIN {X -0.063,Y -591.473,Z 1124.619,A 0.000,B 0.000,C 90.000,E1 327.327} C_DIS
LIN {X 0.225,Y -588.427,Z 1124.614,A 0.000,B 0.000,C 90.000,E1 326.501} C_DIS
LIN {X -0.263,Y -585.512,Z 1124.610,A 0.000,B 0.000,C 90.000,E1 325.881} C_DIS
LIN {X 0.035,Y -582.363,Z 1124.607,A 0.000,B 0.000,C 90.000,E1 325.182} C_DIS
LIN {X -0.090,Y -576.558,Z 1124.601,A 0.000,B 0.000,C 90.000,E1 324.116} C_DIS
LIN {X -0.120,Y -573.375,Z 1124.598,A 0.000,B 0.000,C 90.000,E1 323.577} C_DIS
LIN {X -0.158,Y -568.342,Z 1124.593,A 0.000,B 0.000,C 90.000,E1 322.763} C_DIS
LIN {X -0.134,Y -560.747,Z 1124.587,A 0.000,B 0.000,C 90.000,E1 321.662} C_DIS
LIN {X 0.210,Y -552.396,Z 1124.581,A 0.000,B 0.000,C 90.000,E1 320.517} C_DIS
LIN {X 0.347,Y -543.695,Z 1124.575,A 0.000,B 0.000,C 90.000,E1 319.380} C_DIS
LIN {X -0.011,Y -539.423,Z 1124.571,A 0.000,B 0.000,C 90.000,E1 318.852} C_DIS
LIN {X 0.181,Y -536.406,Z 1124.569,A 0.000,B 0.000,C 90.000,E1 318.405} C_DIS
LIN {X -0.041,Y -533.732,Z 1124.567,A 0.000,B 0.000,C 90.000,E1 318.000} C_DIS
LIN {X 0.244,Y -531.249,Z 1124.564,A 0.000,B 0.000,C 90.000,E1 317.472} C_DIS
LIN {X -0.079,Y -529.619,Z 1124.561,A 0.000,B 0.000,C 90.000,E1 317.025} C_DIS
LIN {X 0.084,Y -529.308,Z 1124.560,A 0.000,B 0.000,C 90.000,E1 316.824} C_DIS
LIN {X 0.212,Y -528.229,Z 1124.558,A 0.000,B 0.000,C 90.000,E1 316.377} C_DIS
LIN {X 0.224,Y -527.878,Z 1124.556,A 0.000,B 0.000,C 90.000,E1 316.053} C_DIS
LIN {X 0.123,Y -526.981,Z 1124.553,A 0.000,B 0.000,C 90.000,E1 315.486} C_DIS
LIN {X -0.239,Y -526.812,Z 1124.551,A 0.000,B 0.000,C 90.000,E1 315.243} C_DIS
LIN {X 0.023,Y -526.096,Z 1124.548,A 0.000,B 0.000,C 90.000,E1 314.636} C_DIS
LIN {X 0.044,Y -525.386,Z 1124.538,A 0.000,B 0.000,C 90.000,E1 312.894} C_DIS
LIN {X 0.054,Y -526.910,Z 1124.514,A 0.000,B 0.000,C 90.000,E1 308.543} C_DIS
LIN {X 0.138,Y -528.513,Z 1124.500,A 0.000,B 0.000,C 90.000,E1 305.931} C_DIS
LIN {X 0.133,Y -529.823,Z 1124.490,A 0.000,B 0.000,C 90.000,E1 304.199} C_DIS
LIN {X -0.175,Y -531.547,Z 1124.477,A 0.000,B 0.000,C 90.000,E1 301.926} C_DIS
LIN {X -0.112,Y -533.584,Z 1124.463,A 0.000,B 0.000,C 90.000,E1 299.333} C_DIS
LIN {X 0.187,Y -534.315,Z 1124.457,A 0.000,B 0.000,C 90.000,E1 298.153} C_DIS
LIN {X 0.247,Y -534.951,Z 1124.450,A 0.000,B 0.000,C 90.000,E1 297.001} C_DIS
LIN {X 0.038,Y -535.447,Z 1124.442,A 0.000,B 0.000,C 90.000,E1 295.591} C_DIS
LIN {X 0.096,Y -535.650,Z 1124.434,A 0.000,B 0.000,C 90.000,E1 294.155} C_DIS
LIN {X 0.089,Y -535.716,Z 1124.423,A 0.000,B 0.000,C 90.000,E1 292.153} C_DIS
LIN {X -0.050,Y -535.706,Z 1124.415,A 0.000,B 0.000,C 90.000,E1 290.737} C_DIS
LIN {X -0.167,Y -535.477,Z 1124.406,A 0.000,B 0.000,C 90.000,E1 289.033} C_DIS
LIN {X 0.011,Y -535.148,Z 1124.398,A 0.000,B 0.000,C 90.000,E1 287.583} C_DIS
LIN {X -0.020,Y -534.833,Z 1124.391,A 0.000,B 0.000,C 90.000,E1 286.441} C_DIS
LIN {X 0.075,Y -533.956,Z 1124.380,A 0.000,B 0.000,C 90.000,E1 284.426} C_DIS
LIN {X 0.138,Y -532.933,Z 1124.369,A 0.000,B 0.000,C 90.000,E1 282.411} C_DIS
LIN {X -0.158,Y -532.194,Z 1124.361,A 0.000,B 0.000,C 90.000,E1 281.007} C_DIS
LIN {X -0.040,Y -531.443,Z 1124.353,A 0.000,B 0.000,C 90.000,E1 279.557} C_DIS
LIN {X 0.103,Y -530.529,Z 1124.344,A 0.000,B 0.000,C 90.000,E1 277.814} C_DIS
LIN {X 0.079,Y -529.432,Z 1124.331,A 0.000,B 0.000,C 90.000,E1 275.511} C_DIS
LIN {X 0.041,Y -528.675,Z 1124.321,A 0.000,B 0.000,C 90.000,E1 273.784} C_DIS
LIN {X -0.093,Y -527.760,Z 1124.310,A 0.000,B 0.000,C 90.000,E1 271.776} C_DIS
LIN {X -0.250,Y -526.964,Z 1124.300,A 0.000,B 0.000,C 90.000,E1 270.057} C_DIS
LIN {X 0.101,Y -526.181,Z 1124.291,A 0.000,B 0.000,C 90.000,E1 268.282} C_DIS
LIN {X -0.020,Y -525.455,Z 1124.282,A 0.000,B 0.000,C 90.000,E1 266.846} C_DIS
LIN {X -0.228,Y -524.171,Z 1124.271,A 0.000,B 0.000,C 90.000,E1 264.837} C_DIS
LIN {X 0.244,Y -523.783,Z 1124.268,A 0.000,B 0.000,C 90.000,E1 264.204} C_DIS
LIN {X 0.136,Y -522.763,Z 1124.262,A 0.000,B 0.000,C 90.000,E1 263.053} C_DIS
LIN {X 0.002,Y -519.982,Z 1124.245,A 0.000,B 0.000,C 90.000,E1 260.151} C_DIS
LIN {X -0.107,Y -518.561,Z 1124.237,A 0.000,B 0.000,C 90.000,E1 258.701} C_DIS
LIN {X -0.037,Y -517.101,Z 1124.229,A 0.000,B 0.000,C 90.000,E1 257.229} C_DIS
LIN {X 0.015,Y -515.713,Z 1124.221,A 0.000,B 0.000,C 90.000,E1 255.755} C_DIS
LIN {X 0.032,Y -514.351,Z 1124.213,A 0.000,B 0.000,C 90.000,E1 254.283} C_DIS
LIN {X -0.118,Y -512.263,Z 1124.201,A 0.000,B 0.000,C 90.000,E1 252.236} C_DIS
LIN {X 0.116,Y -510.726,Z 1124.193,A 0.000,B 0.000,C 90.000,E1 250.732} C_DIS
LIN {X 0.112,Y -508.682,Z 1124.183,A 0.000,B 0.000,C 90.000,E1 248.954} C_DIS
LIN {X -0.038,Y -507.002,Z 1124.175,A 0.000,B 0.000,C 90.000,E1 247.486} C_DIS
LIN {X 0.169,Y -505.046,Z 1124.167,A 0.000,B 0.000,C 90.000,E1 245.973} C_DIS
LIN {X 0.128,Y -502.946,Z 1124.158,A 0.000,B 0.000,C 90.000,E1 244.485} C_DIS
LIN {X 0.084,Y -500.380,Z 1124.148,A 0.000,B 0.000,C 90.000,E1 242.692} C_DIS
LIN {X 0.170,Y -497.993,Z 1124.140,A 0.000,B 0.000,C 90.000,E1 241.179} C_DIS
LIN {X 0.087,Y -494.566,Z 1124.128,A 0.000,B 0.000,C 90.000,E1 239.076} C_DIS
LIN {X 0.157,Y -491.509,Z 1124.118,A 0.000,B 0.000,C 90.000,E1 237.248} C_DIS
LIN {X -0.334,Y -489.447,Z 1124.111,A 0.000,B 0.000,C 90.000,E1 236.087} C_DIS
LIN {X 0.164,Y -486.184,Z 1124.101,A 0.000,B 0.000,C 90.000,E1 234.196} C_DIS
LIN {X -0.133,Y -484.107,Z 1124.094,A 0.000,B 0.000,C 90.000,E1 233.004} C_DIS
LIN {X 0.008,Y -482.439,Z 1124.089,A 0.000,B 0.000,C 90.000,E1 232.065} C_DIS
LIN {X -0.036,Y -478.455,Z 1124.077,A 0.000,B 0.000,C 90.000,E1 229.908} C_DIS
LIN {X 0.238,Y -475.611,Z 1124.069,A 0.000,B 0.000,C 90.000,E1 228.324} C_DIS
LIN {X 0.097,Y -472.737,Z 1124.060,A 0.000,B 0.000,C 90.000,E1 226.782} C_DIS
LIN {X 0.053,Y -468.798,Z 1124.048,A 0.000,B 0.000,C 90.000,E1 224.595} C_DIS
LIN {X 0.178,Y -465.785,Z 1124.037,A 0.000,B 0.000,C 90.000,E1 222.690} C_DIS
LIN {X 0.012,Y -462.422,Z 1124.025,A 0.000,B 0.000,C 90.000,E1 220.496} C_DIS
LIN {X -0.127,Y -458.495,Z 1124.009,A 0.000,B 0.000,C 90.000,E1 217.649} C_DIS
LIN {X -0.075,Y -456.238,Z 1123.998,A 0.000,B 0.000,C 90.000,E1 215.724} C_DIS
LIN {X -0.063,Y -454.312,Z 1123.990,A 0.000,B 0.000,C 90.000,E1 214.119} C_DIS
LIN {X -0.062,Y -451.565,Z 1123.975,A 0.000,B 0.000,C 90.000,E1 211.544} C_DIS
LIN {X -0.044,Y -449.106,Z 1123.957,A 0.000,B 0.000,C 90.000,E1 208.309} C_DIS
LIN {X 0.116,Y -448.397,Z 1123.948,A 0.000,B 0.000,C 90.000,E1 206.668} C_DIS
LIN {X -0.210,Y -448.356,Z 1123.941,A 0.000,B 0.000,C 90.000,E1 205.412} C_DIS
LIN {X 0.066,Y -448.920,Z 1123.934,A 0.000,B 0.000,C 90.000,E1 204.079} C_DIS
LIN {X -0.126,Y -449.838,Z 1123.928,A 0.000,B 0.000,C 90.000,E1 203.131} C_DIS
LIN {X 0.123,Y -452.280,Z 1123.919,A 0.000,B 0.000,C 90.000,E1 201.482} C_DIS
LIN {X -0.087,Y -456.503,Z 1123.909,A 0.000,B 0.000,C 90.000,E1 199.577} C_DIS
LIN {X 0.077,Y -462.053,Z 1123.898,A 0.000,B 0.000,C 90.000,E1 197.638} C_DIS
LIN {X 0.050,Y -472.765,Z 1123.880,A 0.000,B 0.000,C 90.000,E1 194.481} C_DIS
LIN {X 0.136,Y -482.884,Z 1123.866,A 0.000,B 0.000,C 90.000,E1 191.827} C_DIS
LIN {X 0.226,Y -491.611,Z 1123.854,A 0.000,B 0.000,C 90.000,E1 189.670} C_DIS
LIN {X 0.054,Y -499.196,Z 1123.844,A 0.000,B 0.000,C 90.000,E1 187.871} C_DIS
LIN {X -0.147,Y -504.752,Z 1123.836,A 0.000,B 0.000,C 90.000,E1 186.543} C_DIS
LIN {X 0.196,Y -510.265,Z 1123.829,A 0.000,B 0.000,C 90.000,E1 185.163} C_DIS
LIN {X -0.168,Y -516.364,Z 1123.821,A 0.000,B 0.000,C 90.000,E1 183.726} C_DIS
LIN {X 0.018,Y -523.786,Z 1123.811,A 0.000,B 0.000,C 90.000,E1 181.949} C_DIS
LIN {X -0.183,Y -533.594,Z 1123.798,A 0.000,B 0.000,C 90.000,E1 179.656} C_DIS
LIN {X 0.115,Y -540.286,Z 1123.789,A 0.000,B 0.000,C 90.000,E1 178.051} C_DIS
LIN {X -0.241,Y -547.622,Z 1123.780,A 0.000,B 0.000,C 90.000,E1 176.388} C_DIS
LIN {X -0.026,Y -552.480,Z 1123.774,A 0.000,B 0.000,C 90.000,E1 175.241} C_DIS
LIN {X -0.058,Y -559.830,Z 1123.764,A 0.000,B 0.000,C 90.000,E1 173.571} C_DIS
LIN {X -0.098,Y -567.725,Z 1123.754,A 0.000,B 0.000,C 90.000,E1 171.781} C_DIS
LIN {X -0.173,Y -573.106,Z 1123.747,A 0.000,B 0.000,C 90.000,E1 170.557} C_DIS
LIN {X 0.182,Y -578.966,Z 1123.740,A 0.000,B 0.000,C 90.000,E1 169.162} C_DIS
LIN {X 0.057,Y -584.508,Z 1123.732,A 0.000,B 0.000,C 90.000,E1 167.825} C_DIS
LIN {X 0.275,Y -589.961,Z 1123.725,A 0.000,B 0.000,C 90.000,E1 166.464} C_DIS
LIN {X -0.122,Y -595.148,Z 1123.718,A 0.000,B 0.000,C 90.000,E1 165.172} C_DIS
LIN {X -0.284,Y -598.037,Z 1123.713,A 0.000,B 0.000,C 90.000,E1 164.393} C_DIS
LIN {X 0.164,Y -600.870,Z 1123.709,A 0.000,B 0.000,C 90.000,E1 163.559} C_DIS
LIN {X 0.272,Y -605.150,Z 1123.702,A 0.000,B 0.000,C 90.000,E1 162.236} C_DIS
LIN {X 0.184,Y -610.058,Z 1123.693,A 0.000,B 0.000,C 90.000,E1 160.678} C_DIS
LIN {X 0.067,Y -613.853,Z 1123.686,A 0.000,B 0.000,C 90.000,E1 159.390} C_DIS
LIN {X -0.012,Y -618.127,Z 1123.677,A 0.000,B 0.000,C 90.000,E1 157.847} C_DIS
LIN {X 0.245,Y -621.494,Z 1123.670,A 0.000,B 0.000,C 90.000,E1 156.538} C_DIS
LIN {X -0.009,Y -624.782,Z 1123.663,A 0.000,B 0.000,C 90.000,E1 155.281} C_DIS
LIN {X -0.197,Y -628.490,Z 1123.654,A 0.000,B 0.000,C 90.000,E1 153.768} C_DIS
LIN {X -0.074,Y -631.482,Z 1123.647,A 0.000,B 0.000,C 90.000,E1 152.487} C_DIS
LIN {X -0.081,Y -635.334,Z 1123.637,A 0.000,B 0.000,C 90.000,E1 150.717} C_DIS
LIN {X -0.095,Y -638.001,Z 1123.630,A 0.000,B 0.000,C 90.000,E1 149.459} C_DIS
LIN {X -0.071,Y -640.517,Z 1123.623,A 0.000,B 0.000,C 90.000,E1 148.201} C_DIS
LIN {X -0.161,Y -643.372,Z 1123.615,A 0.000,B 0.000,C 90.000,E1 146.707} C_DIS
LIN {X 0.225,Y -645.205,Z 1123.609,A 0.000,B 0.000,C 90.000,E1 145.674} C_DIS
LIN {X -0.372,Y -647.319,Z 1123.603,A 0.000,B 0.000,C 90.000,E1 144.482} C_DIS
LIN {X -0.033,Y -649.451,Z 1123.596,A 0.000,B 0.000,C 90.000,E1 143.210} C_DIS
LIN {X -0.274,Y -652.950,Z 1123.585,A 0.000,B 0.000,C 90.000,E1 141.251} C_DIS
LIN {X -0.004,Y -655.651,Z 1123.576,A 0.000,B 0.000,C 90.000,E1 139.747} C_DIS
LIN {X 0.294,Y -658.912,Z 1123.567,A 0.000,B 0.000,C 90.000,E1 138.000} C_DIS
LIN {X -0.253,Y -660.823,Z 1123.561,A 0.000,B 0.000,C 90.000,E1 137.067} C_DIS
LIN {X 0.122,Y -664.382,Z 1123.552,A 0.000,B 0.000,C 90.000,E1 135.324} C_DIS
LIN {X 0.108,Y -669.384,Z 1123.540,A 0.000,B 0.000,C 90.000,E1 133.137} C_DIS
LIN {X -0.209,Y -674.034,Z 1123.529,A 0.000,B 0.000,C 90.000,E1 131.229} C_DIS
LIN {X -0.044,Y -676.928,Z 1123.522,A 0.000,B 0.000,C 90.000,E1 130.011} C_DIS
LIN {X -0.056,Y -682.460,Z 1123.510,A 0.000,B 0.000,C 90.000,E1 127.855} C_DIS
LIN {X -0.070,Y -685.511,Z 1123.504,A 0.000,B 0.000,C 90.000,E1 126.664} C_DIS
LIN {X 0.008,Y -689.053,Z 1123.496,A 0.000,B 0.000,C 90.000,E1 125.231} C_DIS
LIN {X 0.322,Y -692.567,Z 1123.488,A 0.000,B 0.000,C 90.000,E1 123.785} C_DIS
LIN {X -0.254,Y -695.912,Z 1123.480,A 0.000,B 0.000,C 90.000,E1 122.418} C_DIS
LIN {X 0.162,Y -698.503,Z 1123.474,A 0.000,B 0.000,C 90.000,E1 121.209} C_DIS
LIN {X 0.353,Y -700.193,Z 1123.468,A 0.000,B 0.000,C 90.000,E1 120.256} C_DIS
LIN {X 0.139,Y -702.571,Z 1123.460,A 0.000,B 0.000,C 90.000,E1 118.871} C_DIS
LIN {X 0.024,Y -703.775,Z 1123.457,A 0.000,B 0.000,C 90.000,E1 118.180} C_DIS
LIN {X -0.082,Y -704.876,Z 1123.451,A 0.000,B 0.000,C 90.000,E1 117.257} C_DIS
LIN {X 0.153,Y -705.445,Z 1123.448,A 0.000,B 0.000,C 90.000,E1 116.539} C_DIS
LIN {X -0.279,Y -706.193,Z 1123.441,A 0.000,B 0.000,C 90.000,E1 115.412} C_DIS
LIN {X 0.015,Y -706.318,Z 1123.440,A 0.000,B 0.000,C 90.000,E1 115.155} C_DIS
LIN {X -0.043,Y -706.117,Z 1123.437,A 0.000,B 0.000,C 90.000,E1 114.695} C_DIS
LIN {X -0.045,Y -705.898,Z 1123.436,A 0.000,B 0.000,C 90.000,E1 114.463} C_DIS
LIN {X -0.109,Y -705.114,Z 1123.433,A 0.000,B 0.000,C 90.000,E1 114.003} C_DIS
LIN {X -0.108,Y -704.302,Z 1123.432,A 0.000,B 0.000,C 90.000,E1 113.770} C_DIS
LIN {X 0.180,Y -702.307,Z 1123.429,A 0.000,B 0.000,C 90.000,E1 113.281} C_DIS
LIN {X -0.325,Y -701.444,Z 1123.429,A 0.000,B 0.000,C 90.000,E1 113.206} C_DIS
LIN {X -0.057,Y -697.060,Z 1123.426,A 0.000,B 0.000,C 90.000,E1 112.717} C_DIS
LIN {X 0.073,Y -695.487,Z 1123.426,A 0.000,B 0.000,C 90.000,E1 112.589} C_DIS
LIN {X -0.253,Y -693.202,Z 1123.425,A 0.000,B 0.000,C 90.000,E1 112.514} C_DIS
LIN {X -0.135,Y -687.053,Z 1123.424,A 0.000,B 0.000,C 90.000,E1 112.280} C_DIS
LIN {X 0.022,Y -684.967,Z 1123.423,A 0.000,B 0.000,C 90.000,E1 112.206} C_DIS
LIN {X 0.146,Y -676.182,Z 1123.423,A 0.000,B 0.000,C 90.000,E1 112.099} C_DIS
LIN {X 0.095,Y -603.260,Z 1123.423,A 0.000,B 0.000,C 90.000,E1 112.099} C_DIS
LIN {X 0.212,Y -600.166,Z 1123.422,A 0.000,B 0.000,C 90.000,E1 111.897} C_DIS
LIN {X -0.153,Y -595.652,Z 1123.420,A 0.000,B 0.000,C 90.000,E1 111.589} C_DIS
LIN {X -0.200,Y -579.583,Z 1123.412,A 0.000,B 0.000,C 90.000,E1 110.174} C_DIS
LIN {X -0.168,Y -575.404,Z 1123.410,A 0.000,B 0.000,C 90.000,E1 109.812} C_DIS
LIN {X 0.141,Y -569.461,Z 1123.407,A 0.000,B 0.000,C 90.000,E1 109.322} C_DIS
LIN {X -0.215,Y -564.561,Z 1123.406,A 0.000,B 0.000,C 90.000,E1 109.033} C_DIS
LIN {X 0.316,Y -561.485,Z 1123.405,A 0.000,B 0.000,C 90.000,E1 108.779} C_DIS
LIN {X 0.082,Y -554.785,Z 1123.402,A 0.000,B 0.000,C 90.000,E1 108.417} C_DIS
LIN {X -0.229,Y -550.301,Z 1123.401,A 0.000,B 0.000,C 90.000,E1 108.127} C_DIS
LIN {X -0.113,Y -549.196,Z 1123.400,A 0.000,B 0.000,C 90.000,E1 107.928} C_DIS
LIN {X -0.156,Y -549.181,Z 1123.400,A 0.000,B 0.000,C 90.000,E1 107.928} C_DIS
LIN {X 0.164,Y -548.893,Z 1123.398,A 0.000,B 0.000,C 90.000,E1 107.583} C_DIS
LIN {X -0.214,Y -550.104,Z 1123.387,A 0.000,B 0.000,C 90.000,E1 105.607} C_DIS
LIN {X 0.176,Y -551.355,Z 1123.377,A 0.000,B 0.000,C 90.000,E1 103.883} C_DIS
LIN {X 0.039,Y -553.246,Z 1123.365,A 0.000,B 0.000,C 90.000,E1 101.658} C_DIS
LIN {X -0.177,Y -555.036,Z 1123.354,A 0.000,B 0.000,C 90.000,E1 99.726} C_DIS
LIN {X -0.258,Y -556.333,Z 1123.346,A 0.000,B 0.000,C 90.000,E1 98.341} C_DIS
LIN {X -0.170,Y -557.915,Z 1123.337,A 0.000,B 0.000,C 90.000,E1 96.663} C_DIS
LIN {X -0.118,Y -559.519,Z 1123.328,A 0.000,B 0.000,C 90.000,E1 94.992} C_DIS
LIN {X -0.169,Y -560.644,Z 1123.320,A 0.000,B 0.000,C 90.000,E1 93.612} C_DIS
LIN {X -0.237,Y -561.643,Z 1123.312,A 0.000,B 0.000,C 90.000,E1 92.236} C_DIS
LIN {X 0.275,Y -562.512,Z 1123.305,A 0.000,B 0.000,C 90.000,E1 90.802} C_DIS
LIN {X 0.226,Y -563.333,Z 1123.297,A 0.000,B 0.000,C 90.000,E1 89.427} C_DIS
LIN {X -0.146,Y -564.407,Z 1123.286,A 0.000,B 0.000,C 90.000,E1 87.535} C_DIS
LIN {X 0.097,Y -565.318,Z 1123.276,A 0.000,B 0.000,C 90.000,E1 85.584} C_DIS
LIN {X 0.304,Y -566.029,Z 1123.266,A 0.000,B 0.000,C 90.000,E1 83.913} C_DIS
LIN {X 0.129,Y -566.840,Z 1123.256,A 0.000,B 0.000,C 90.000,E1 82.008} C_DIS
LIN {X 0.047,Y -567.624,Z 1123.245,A 0.000,B 0.000,C 90.000,E1 80.095} C_DIS
LIN {X 0.252,Y -568.539,Z 1123.233,A 0.000,B 0.000,C 90.000,E1 77.881} C_DIS
LIN {X -0.197,Y -569.325,Z 1123.224,A 0.000,B 0.000,C 90.000,E1 76.284} C_DIS
LIN {X 0.255,Y -570.898,Z 1123.208,A 0.000,B 0.000,C 90.000,E1 73.504} C_DIS
LIN {X -0.187,Y -572.261,Z 1123.198,A 0.000,B 0.000,C 90.000,E1 71.638} C_DIS
LIN {X 0.120,Y -574.327,Z 1123.184,A 0.000,B 0.000,C 90.000,E1 69.156} C_DIS
LIN {X -0.173,Y -576.058,Z 1123.174,A 0.000,B 0.000,C 90.000,E1 67.283} C_DIS
LIN {X 0.041,Y -577.041,Z 1123.168,A 0.000,B 0.000,C 90.000,E1 66.177} C_DIS
LIN {X 0.199,Y -578.422,Z 1123.159,A 0.000,B 0.000,C 90.000,E1 64.537} C_DIS
LIN {X 0.003,Y -579.575,Z 1123.151,A 0.000,B 0.000,C 90.000,E1 63.204} C_DIS
LIN {X 0.083,Y -580.613,Z 1123.144,A 0.000,B 0.000,C 90.000,E1 61.847} C_DIS
LIN {X -0.317,Y -581.956,Z 1123.133,A 0.000,B 0.000,C 90.000,E1 59.999} C_DIS
LIN {X 0.251,Y -582.961,Z 1123.124,A 0.000,B 0.000,C 90.000,E1 58.329} C_DIS
LIN {X -0.292,Y -584.006,Z 1123.114,A 0.000,B 0.000,C 90.000,E1 56.501} C_DIS
LIN {X -0.163,Y -585.003,Z 1123.103,A 0.000,B 0.000,C 90.000,E1 54.609} C_DIS
LIN {X -0.014,Y -585.902,Z 1123.093,A 0.000,B 0.000,C 90.000,E1 52.718} C_DIS
LIN {X 0.091,Y -586.212,Z 1123.089,A 0.000,B 0.000,C 90.000,E1 51.904} C_DIS
LIN {X 0.131,Y -586.675,Z 1123.081,A 0.000,B 0.000,C 90.000,E1 50.561} C_DIS
LIN {X 0.181,Y -586.794,Z 1123.074,A 0.000,B 0.000,C 90.000,E1 49.218} C_DIS
LIN {X -0.212,Y -586.712,Z 1123.066,A 0.000,B 0.000,C 90.000,E1 47.919} C_DIS
LIN {X 0.214,Y -586.429,Z 1123.059,A 0.000,B 0.000,C 90.000,E1 46.539} C_DIS
LIN {X -0.219,Y -585.974,Z 1123.051,A 0.000,B 0.000,C 90.000,E1 45.243} C_DIS
LIN {X 0.171,Y -585.232,Z 1123.044,A 0.000,B 0.000,C 90.000,E1 43.866} C_DIS
LIN {X 0.137,Y -584.130,Z 1123.036,A 0.000,B 0.000,C 90.000,E1 42.528} C_DIS
LIN {X -0.044,Y -582.999,Z 1123.030,A 0.000,B 0.000,C 90.000,E1 41.472} C_DIS
LIN {X 0.142,Y -581.691,Z 1123.024,A 0.000,B 0.000,C 90.000,E1 40.378} C_DIS
LIN {X -0.075,Y -580.185,Z 1123.018,A 0.000,B 0.000,C 90.000,E1 39.322} C_DIS
LIN {X -0.226,Y -578.327,Z 1123.012,A 0.000,B 0.000,C 90.000,E1 38.257} C_DIS
LIN {X -0.039,Y -576.322,Z 1123.006,A 0.000,B 0.000,C 90.000,E1 37.156} C_DIS
LIN {X -0.042,Y -574.379,Z 1123.002,A 0.000,B 0.000,C 90.000,E1 36.343} C_DIS
LIN {X 0.197,Y -571.512,Z 1122.996,A 0.000,B 0.000,C 90.000,E1 35.231} C_DIS
LIN {X 0.271,Y -568.866,Z 1122.991,A 0.000,B 0.000,C 90.000,E1 34.405} C_DIS
LIN {X -0.269,Y -566.968,Z 1122.988,A 0.000,B 0.000,C 90.000,E1 33.913} C_DIS
LIN {X -0.350,Y -564.877,Z 1122.985,A 0.000,B 0.000,C 90.000,E1 33.372} C_DIS
LIN {X 0.132,Y -561.380,Z 1122.981,A 0.000,B 0.000,C 90.000,E1 32.498} C_DIS
LIN {X 0.018,Y -558.872,Z 1122.978,A 0.000,B 0.000,C 90.000,E1 31.957} C_DIS
LIN {X 0.061,Y -555.486,Z 1122.974,A 0.000,B 0.000,C 90.000,E1 31.258} C_DIS
LIN {X -0.215,Y -551.858,Z 1122.970,A 0.000,B 0.000,C 90.000,E1 30.590} C_DIS
LIN {X -0.018,Y -546.425,Z 1122.964,A 0.000,B 0.000,C 90.000,E1 29.589} C_DIS
LIN {X -0.038,Y -543.076,Z 1122.961,A 0.000,B 0.000,C 90.000,E1 29.027} C_DIS
LIN {X 0.185,Y -539.469,Z 1122.958,A 0.000,B 0.000,C 90.000,E1 28.437} C_DIS
LIN {X -0.232,Y -534.653,Z 1122.954,A 0.000,B 0.000,C 90.000,E1 27.769} C_DIS
LIN {X 0.252,Y -529.418,Z 1122.950,A 0.000,B 0.000,C 90.000,E1 27.001} C_DIS
LIN {X -0.019,Y -523.688,Z 1122.946,A 0.000,B 0.000,C 90.000,E1 26.309} C_DIS
LIN {X 0.197,Y -516.298,Z 1122.941,A 0.000,B 0.000,C 90.000,E1 25.412} C_DIS
LIN {X 0.020,Y -511.014,Z 1122.938,A 0.000,B 0.000,C 90.000,E1 24.847} C_DIS
LIN {X 0.033,Y -504.487,Z 1122.934,A 0.000,B 0.000,C 90.000,E1 24.155} C_DIS
LIN {X -0.073,Y -497.582,Z 1122.930,A 0.000,B 0.000,C 90.000,E1 23.462} C_DIS
LIN {X 0.175,Y -489.496,Z 1122.926,A 0.000,B 0.000,C 90.000,E1 22.642} C_DIS
LIN {X -0.115,Y -481.150,Z 1122.922,A 0.000,B 0.000,C 90.000,E1 21.897} C_DIS
LIN {X -0.057,Y -472.235,Z 1122.917,A 0.000,B 0.000,C 90.000,E1 21.099} C_DIS
LIN {X -0.021,Y -461.789,Z 1122.912,A 0.000,B 0.000,C 90.000,E1 20.174} C_DIS
LIN {X -0.238,Y -445.377,Z 1122.904,A 0.000,B 0.000,C 90.000,E1 18.725} C_DIS
LIN {X 0.059,Y -429.677,Z 1122.895,A 0.000,B 0.000,C 90.000,E1 17.149} C_DIS
LIN {X 0.059,Y -417.121,Z 1122.888,A 0.000,B 0.000,C 90.000,E1 15.788} C_DIS
LIN {X 0.062,Y -409.103,Z 1122.882,A 0.000,B 0.000,C 90.000,E1 14.828} C_DIS
LIN {X 0.083,Y -400.255,Z 1122.876,A 0.000,B 0.000,C 90.000,E1 13.647} C_DIS
LIN {X 0.118,Y -399.126,Z 1122.875,A 0.000,B 0.000,C 90.000,E1 13.480} C_DIS
LIN {X 0.166,Y -395.131,Z 1122.871,A 0.000,B 0.000,C 90.000,E1 12.771} C_DIS
LIN {X 0.099,Y -393.440,Z 1122.869,A 0.000,B 0.000,C 90.000,E1 12.355} C_DIS
LIN {X 0.039,Y -392.916,Z 1122.868,A 0.000,B 0.000,C 90.000,E1 12.187} C_DIS
LIN {X 0.063,Y -392.259,Z 1122.866,A 0.000,B 0.000,C 90.000,E1 11.827} C_DIS
LIN {X -0.047,Y -392.101,Z 1122.863,A 0.000,B 0.000,C 90.000,E1 11.299} C_DIS
LIN {X -0.108,Y -392.189,Z 1122.862,A 0.000,B 0.000,C 90.000,E1 11.130} C_DIS
LIN {X -0.063,Y -393.527,Z 1122.857,A 0.000,B 0.000,C 90.000,E1 10.197} C_DIS
LIN {X -0.143,Y -394.937,Z 1122.853,A 0.000,B 0.000,C 90.000,E1 9.500} C_DIS
LIN {X -0.010,Y -403.496,Z 1122.835,A 0.000,B 0.000,C 90.000,E1 6.315} C_DIS
LIN {X -0.018,Y -404.532,Z 1122.833,A 0.000,B 0.000,C 90.000,E1 5.967} C_DIS
LIN {X -0.062,Y -407.215,Z 1122.829,A 0.000,B 0.000,C 90.000,E1 5.277} C_DIS
LIN {X -0.007,Y -411.681,Z 1122.826,A 0.000,B 0.000,C 90.000,E1 4.645} C_DIS
LIN {X 0.106,Y -416.730,Z 1122.823,A 0.000,B 0.000,C 90.000,E1 4.188} C_DIS
LIN {X 0.079,Y -427.576,Z 1122.819,A 0.000,B 0.000,C 90.000,E1 3.440} C_DIS
LIN {X -0.211,Y -447.204,Z 1122.812,A 0.000,B 0.000,C 90.000,E1 2.121} C_DIS
LIN {X -0.097,Y -461.950,Z 1122.806,A 0.000,B 0.000,C 90.000,E1 1.146} C_DIS
LIN {X -0.047,Y -473.343,Z 1122.802,A 0.000,B 0.000,C 90.000,E1 0.401} C_DIS
LIN {X -0.220,Y -484.084,Z 1122.798,A 0.000,B 0.000,C 90.000,E1 359.714} C_DIS
LIN {X 0.037,Y -491.825,Z 1122.795,A 0.000,B 0.000,C 90.000,E1 359.141} C_DIS
LIN {X 0.203,Y -497.817,Z 1122.793,A 0.000,B 0.000,C 90.000,E1 358.682} C_DIS
LIN {X 0.095,Y -503.880,Z 1122.790,A 0.000,B 0.000,C 90.000,E1 358.224} C_DIS
LIN {X -0.128,Y -509.860,Z 1122.788,A 0.000,B 0.000,C 90.000,E1 357.764} C_DIS
LIN {X -0.111,Y -516.845,Z 1122.784,A 0.000,B 0.000,C 90.000,E1 357.135} C_DIS
LIN {X -0.073,Y -524.938,Z 1122.780,A 0.000,B 0.000,C 90.000,E1 356.331} C_DIS
LIN {X -0.167,Y -531.353,Z 1122.776,A 0.000,B 0.000,C 90.000,E1 355.641} C_DIS
LIN {X 0.144,Y -537.083,Z 1122.772,A 0.000,B 0.000,C 90.000,E1 354.894} C_DIS
LIN {X 0.190,Y -541.321,Z 1122.769,A 0.000,B 0.000,C 90.000,E1 354.318} C_DIS
LIN {X 0.005,Y -546.113,Z 1122.765,A 0.000,B 0.000,C 90.000,E1 353.628} C_DIS
LIN {X -0.077,Y -550.379,Z 1122.761,A 0.000,B 0.000,C 90.000,E1 352.932} C_DIS
LIN {X 0.066,Y -553.577,Z 1122.758,A 0.000,B 0.000,C 90.000,E1 352.356} C_DIS
LIN {X 0.056,Y -557.168,Z 1122.754,A 0.000,B 0.000,C 90.000,E1 351.659} C_DIS
LIN {X 0.243,Y -559.702,Z 1122.751,A 0.000,B 0.000,C 90.000,E1 351.084} C_DIS
LIN {X -0.020,Y -562.060,Z 1122.748,A 0.000,B 0.000,C 90.000,E1 350.557} C_DIS
LIN {X -0.203,Y -565.311,Z 1122.743,A 0.000,B 0.000,C 90.000,E1 349.746} C_DIS
LIN {X -0.074,Y -569.334,Z 1122.737,A 0.000,B 0.000,C 90.000,E1 348.634} C_DIS
LIN {X 0.116,Y -572.930,Z 1122.731,A 0.000,B 0.000,C 90.000,E1 347.521} C_DIS
LIN {X -0.204,Y -576.301,Z 1122.725,A 0.000,B 0.000,C 90.000,E1 346.464} C_DIS
LIN {X -0.126,Y -580.188,Z 1122.717,A 0.000,B 0.000,C 90.000,E1 345.102} C_DIS
LIN {X -0.317,Y -584.592,Z 1122.708,A 0.000,B 0.000,C 90.000,E1 343.504} C_DIS
LIN {X 0.058,Y -588.023,Z 1122.701,A 0.000,B 0.000,C 90.000,E1 342.127} C_DIS
LIN {X 0.251,Y -590.586,Z 1122.695,A 0.000,B 0.000,C 90.000,E1 341.040} C_DIS
LIN {X -0.195,Y -593.538,Z 1122.688,A 0.000,B 0.000,C 90.000,E1 339.752} C_DIS
LIN {X -0.034,Y -596.136,Z 1122.680,A 0.000,B 0.000,C 90.000,E1 338.411} C_DIS
LIN {X 0.329,Y -597.081,Z 1122.677,A 0.000,B 0.000,C 90.000,E1 337.847} C_DIS
LIN {X -0.164,Y -598.259,Z 1122.673,A 0.000,B 0.000,C 90.000,E1 337.102} C_DIS
LIN {X -0.259,Y -599.807,Z 1122.665,A 0.000,B 0.000,C 90.000,E1 335.793} C_DIS
LIN {X 0.063,Y -600.585,Z 1122.661,A 0.000,B 0.000,C 90.000,E1 334.973} C_DIS
LIN {X -0.148,Y -601.100,Z 1122.657,A 0.000,B 0.000,C 90.000,E1 334.204} C_DIS
LIN {X 0.186,Y -601.372,Z 1122.652,A 0.000,B 0.000,C 90.000,E1 333.384} C_DIS
LIN {X -0.018,Y -601.386,Z 1122.648,A 0.000,B 0.000,C 90.000,E1 332.615} C_DIS
LIN {X -0.225,Y -601.196,Z 1122.644,A 0.000,B 0.000,C 90.000,E1 331.847} C_DIS
LIN {X -0.150,Y -600.650,Z 1122.639,A 0.000,B 0.000,C 90.000,E1 331.051} C_DIS
LIN {X -0.074,Y -599.710,Z 1122.635,A 0.000,B 0.000,C 90.000,E1 330.255} C_DIS
LIN {X -0.230,Y -598.873,Z 1122.632,A 0.000,B 0.000,C 90.000,E1 329.744} C_DIS
LIN {X 0.044,Y -596.649,Z 1122.626,A 0.000,B 0.000,C 90.000,E1 328.663} C_DIS
LIN {X 0.074,Y -594.442,Z 1122.622,A 0.000,B 0.000,C 90.000,E1 327.867} C_DIS
LIN {X -0.102,Y -591.807,Z 1122.617,A 0.000,B 0.000,C 90.000,E1 327.089} C_DIS
LIN {X -0.007,Y -589.805,Z 1122.614,A 0.000,B 0.000,C 90.000,E1 326.548} C_DIS
LIN {X -0.061,Y -586.447,Z 1122.610,A 0.000,B 0.000,C 90.000,E1 325.754} C_DIS
LIN {X -0.307,Y -582.741,Z 1122.605,A 0.000,B 0.000,C 90.000,E1 324.975} C_DIS
LIN {X -0.036,Y -579.324,Z 1122.602,A 0.000,B 0.000,C 90.000,E1 324.276} C_DIS
LIN {X -0.263,Y -575.625,Z 1122.598,A 0.000,B 0.000,C 90.000,E1 323.623} C_DIS
LIN {X 0.041,Y -572.534,Z 1122.595,A 0.000,B 0.000,C 90.000,E1 323.050} C_DIS
LIN {X 0.319,Y -569.237,Z 1122.592,A 0.000,B 0.000,C 90.000,E1 322.477} C_DIS
LIN {X -0.108,Y -563.830,Z 1122.587,A 0.000,B 0.000,C 90.000,E1 321.698} C_DIS
LIN {X 0.001,Y -561.980,Z 1122.586,A 0.000,B 0.000,C 90.000,E1 321.412} C_DIS
LIN {X 0.055,Y -556.188,Z 1122.581,A 0.000,B 0.000,C 90.000,E1 320.598} C_DIS
LIN {X -0.222,Y -552.160,Z 1122.578,A 0.000,B 0.000,C 90.000,E1 320.070} C_DIS
LIN {X -0.320,Y -547.099,Z 1122.574,A 0.000,B 0.000,C 90.000,E1 319.380} C_DIS
LIN {X -0.249,Y -538.420,Z 1122.568,A 0.000,B 0.000,C 90.000,E1 318.243} C_DIS
LIN {X -0.060,Y -535.667,Z 1122.566,A 0.000,B 0.000,C 90.000,E1 317.796} C_DIS
LIN {X -0.190,Y -533.446,Z 1122.563,A 0.000,B 0.000,C 90.000,E1 317.391} C_DIS
LIN {X -0.008,Y -531.989,Z 1122.561,A 0.000,B 0.000,C 90.000,E1 316.986} C_DIS
LIN {X -0.030,Y -530.714,Z 1122.559,A 0.000,B 0.000,C 90.000,E1 316.701} C_DIS
LIN {X 0.274,Y -529.789,Z 1122.557,A 0.000,B 0.000,C 90.000,E1 316.215} C_DIS
LIN {X -0.142,Y -528.927,Z 1122.555,A 0.000,B 0.000,C 90.000,E1 315.972} C_DIS
LIN {X -0.222,Y -527.218,Z 1122.549,A 0.000,B 0.000,C 90.000,E1 314.919} C_DIS
LIN {X 0.100,Y -526.828,Z 1122.548,A 0.000,B 0.000,C 90.000,E1 314.595} C_DIS
LIN {X -0.168,Y -525.914,Z 1122.540,A 0.000,B 0.000,C 90.000,E1 313.176} C_DIS
LIN {X -0.184,Y -525.940,Z 1122.529,A 0.000,B 0.000,C 90.000,E1 311.148} C_DIS
LIN {X -0.212,Y -527.165,Z 1122.514,A 0.000,B 0.000,C 90.000,E1 308.543} C_DIS
LIN {X -0.120,Y -528.769,Z 1122.500,A 0.000,B 0.000,C 90.000,E1 305.931} C_DIS
LIN {X -0.120,Y -530.070,Z 1122.490,A 0.000,B 0.000,C 90.000,E1 304.199} C_DIS
LIN {X 0.031,Y -531.796,Z 1122.477,A 0.000,B 0.000,C 90.000,E1 301.878} C_DIS
LIN {X -0.060,Y -533.617,Z 1122.464,A 0.000,B 0.000,C 90.000,E1 299.589} C_DIS
LIN {X -0.017,Y -534.397,Z 1122.458,A 0.000,B 0.000,C 90.000,E1 298.437} C_DIS
LIN {X 0.015,Y -535.195,Z 1122.450,A 0.000,B 0.000,C 90.000,E1 297.001} C_DIS
LIN {X 0.090,Y -535.619,Z 1122.444,A 0.000,B 0.000,C 90.000,E1 295.848} C_DIS
LIN {X 0.092,Y -535.928,Z 1122.434,A 0.000,B 0.000,C 90.000,E1 294.131} C_DIS
LIN {X -0.127,Y -536.009,Z 1122.423,A 0.000,B 0.000,C 90.000,E1 292.153} C_DIS
LIN {X -0.260,Y -536.014,Z 1122.415,A 0.000,B 0.000,C 90.000,E1 290.737} C_DIS
LIN {X 0.311,Y -535.784,Z 1122.406,A 0.000,B 0.000,C 90.000,E1 288.960} C_DIS
LIN {X -0.186,Y -535.472,Z 1122.398,A 0.000,B 0.000,C 90.000,E1 287.583} C_DIS
LIN {X -0.212,Y -535.131,Z 1122.391,A 0.000,B 0.000,C 90.000,E1 286.441} C_DIS
LIN {X -0.205,Y -534.508,Z 1122.383,A 0.000,B 0.000,C 90.000,E1 285.009} C_DIS
LIN {X 0.121,Y -533.998,Z 1122.377,A 0.000,B 0.000,C 90.000,E1 283.828} C_DIS
LIN {X -0.037,Y -533.274,Z 1122.369,A 0.000,B 0.000,C 90.000,E1 282.411} C_DIS
LIN {X 0.196,Y -532.533,Z 1122.361,A 0.000,B 0.000,C 90.000,E1 280.950} C_DIS
LIN {X -0.202,Y -531.785,Z 1122.353,A 0.000,B 0.000,C 90.000,E1 279.557} C_DIS
LIN {X -0.087,Y -531.050,Z 1122.345,A 0.000,B 0.000,C 90.000,E1 278.106} C_DIS
LIN {X -0.036,Y -529.935,Z 1122.332,A 0.000,B 0.000,C 90.000,E1 275.796} C_DIS
LIN {X -0.105,Y -529.174,Z 1122.323,A 0.000,B 0.000,C 90.000,E1 274.073} C_DIS
LIN {X -0.188,Y -528.358,Z 1122.313,A 0.000,B 0.000,C 90.000,E1 272.350} C_DIS
LIN {X 0.259,Y -527.843,Z 1122.307,A 0.000,B 0.000,C 90.000,E1 271.146} C_DIS
LIN {X 0.107,Y -527.086,Z 1122.297,A 0.000,B 0.000,C 90.000,E1 269.427} C_DIS
LIN {X -0.021,Y -526.406,Z 1122.289,A 0.000,B 0.000,C 90.000,E1 267.993} C_DIS
LIN {X -0.157,Y -525.616,Z 1122.281,A 0.000,B 0.000,C 90.000,E1 266.560} C_DIS
LIN {X 0.202,Y -524.337,Z 1122.270,A 0.000,B 0.000,C 90.000,E1 264.489} C_DIS
LIN {X 0.108,Y -523.362,Z 1122.263,A 0.000,B 0.000,C 90.000,E1 263.337} C_DIS
LIN {X -0.077,Y -521.319,Z 1122.252,A 0.000,B 0.000,C 90.000,E1 261.319} C_DIS
LIN {X -0.072,Y -520.307,Z 1122.245,A 0.000,B 0.000,C 90.000,E1 260.151} C_DIS
LIN {X -0.179,Y -518.610,Z 1122.236,A 0.000,B 0.000,C 90.000,E1 258.409} C_DIS
LIN {X -0.097,Y -517.487,Z 1122.229,A 0.000,B 0.000,C 90.000,E1 257.229} C_DIS
LIN {X -0.039,Y -516.060,Z 1122.221,A 0.000,B 0.000,C 90.000,E1 255.755} C_DIS
LIN {X -0.016,Y -514.670,Z 1122.213,A 0.000,B 0.000,C 90.000,E1 254.283} C_DIS
LIN {X -0.157,Y -512.588,Z 1122.201,A 0.000,B 0.000,C 90.000,E1 252.236} C_DIS
LIN {X 0.084,Y -511.037,Z 1122.193,A 0.000,B 0.000,C 90.000,E1 250.732} C_DIS
LIN {X 0.087,Y -508.968,Z 1122.183,A 0.000,B 0.000,C 90.000,E1 248.954} C_DIS
LIN {X -0.058,Y -507.314,Z 1122.175,A 0.000,B 0.000,C 90.000,E1 247.486} C_DIS
LIN {X 0.154,Y -505.377,Z 1122.167,A 0.000,B 0.000,C 90.000,E1 245.973} C_DIS
LIN {X -0.039,Y -502.789,Z 1122.157,A 0.000,B 0.000,C 90.000,E1 244.204} C_DIS
LIN {X 0.083,Y -500.617,Z 1122.148,A 0.000,B 0.000,C 90.000,E1 242.692} C_DIS
LIN {X 0.172,Y -498.244,Z 1122.140,A 0.000,B 0.000,C 90.000,E1 241.179} C_DIS
LIN {X 0.095,Y -494.799,Z 1122.128,A 0.000,B 0.000,C 90.000,E1 239.076} C_DIS
LIN {X 0.171,Y -491.751,Z 1122.118,A 0.000,B 0.000,C 90.000,E1 237.248} C_DIS
LIN {X -0.072,Y -489.089,Z 1122.110,A 0.000,B 0.000,C 90.000,E1 235.754} C_DIS
LIN {X 0.186,Y -486.410,Z 1122.101,A 0.000,B 0.000,C 90.000,E1 234.196} C_DIS
LIN {X 0.009,Y -483.710,Z 1122.093,A 0.000,B 0.000,C 90.000,E1 232.683} C_DIS
LIN {X -0.032,Y -481.409,Z 1122.086,A 0.000,B 0.000,C 90.000,E1 231.457} C_DIS
LIN {X -0.204,Y -478.038,Z 1122.076,A 0.000,B 0.000,C 90.000,E1 229.622} C_DIS
LIN {X 0.057,Y -475.138,Z 1122.067,A 0.000,B 0.000,C 90.000,E1 228.038} C_DIS
LIN {X 0.226,Y -472.225,Z 1122.058,A 0.000,B 0.000,C 90.000,E1 226.458} C_DIS
LIN {X 0.089,Y -468.852,Z 1122.048,A 0.000,B 0.000,C 90.000,E1 224.595} C_DIS
LIN {X 0.215,Y -465.821,Z 1122.037,A 0.000,B 0.000,C 90.000,E1 222.690} C_DIS
LIN {X 0.094,Y -461.911,Z 1122.023,A 0.000,B 0.000,C 90.000,E1 220.172} C_DIS
LIN {X -0.092,Y -458.347,Z 1122.009,A 0.000,B 0.000,C 90.000,E1 217.649} C_DIS
LIN {X 0.226,Y -456.418,Z 1122.000,A 0.000,B 0.000,C 90.000,E1 216.011} C_DIS
LIN {X 0.242,Y -454.475,Z 1121.991,A 0.000,B 0.000,C 90.000,E1 214.405} C_DIS
LIN {X -0.135,Y -451.501,Z 1121.977,A 0.000,B 0.000,C 90.000,E1 211.878} C_DIS
LIN {X 0.092,Y -448.722,Z 1121.959,A 0.000,B 0.000,C 90.000,E1 208.615} C_DIS
LIN {X 0.102,Y -447.620,Z 1121.948,A 0.000,B 0.000,C 90.000,E1 206.668} C_DIS
LIN {X -0.236,Y -447.468,Z 1121.941,A 0.000,B 0.000,C 90.000,E1 205.412} C_DIS
LIN {X 0.025,Y -447.894,Z 1121.934,A 0.000,B 0.000,C 90.000,E1 204.079} C_DIS
LIN {X 0.234,Y -448.755,Z 1121.928,A 0.000,B 0.000,C 90.000,E1 203.078} C_DIS
LIN {X -0.135,Y -450.049,Z 1121.923,A 0.000,B 0.000,C 90.000,E1 202.153} C_DIS
LIN {X 0.095,Y -451.685,Z 1121.918,A 0.000,B 0.000,C 90.000,E1 201.153} C_DIS
LIN {X -0.192,Y -455.283,Z 1121.909,A 0.000,B 0.000,C 90.000,E1 199.577} C_DIS
LIN {X 0.034,Y -459.850,Z 1121.900,A 0.000,B 0.000,C 90.000,E1 197.946} C_DIS
LIN {X 0.054,Y -470.539,Z 1121.882,A 0.000,B 0.000,C 90.000,E1 194.773} C_DIS
LIN {X 0.177,Y -481.326,Z 1121.867,A 0.000,B 0.000,C 90.000,E1 191.951} C_DIS
LIN {X -0.244,Y -490.147,Z 1121.855,A 0.000,B 0.000,C 90.000,E1 189.849} C_DIS
LIN {X 0.046,Y -497.804,Z 1121.844,A 0.000,B 0.000,C 90.000,E1 187.992} C_DIS
LIN {X 0.148,Y -502.805,Z 1121.838,A 0.000,B 0.000,C 90.000,E1 186.777} C_DIS
LIN {X -0.100,Y -509.627,Z 1121.829,A 0.000,B 0.000,C 90.000,E1 185.163} C_DIS
LIN {X 0.184,Y -517.611,Z 1121.818,A 0.000,B 0.000,C 90.000,E1 183.212} C_DIS
LIN {X 0.185,Y -524.483,Z 1121.809,A 0.000,B 0.000,C 90.000,E1 181.604} C_DIS
LIN {X 0.264,Y -533.765,Z 1121.797,A 0.000,B 0.000,C 90.000,E1 179.427} C_DIS
LIN {X -0.244,Y -539.909,Z 1121.789,A 0.000,B 0.000,C 90.000,E1 178.051} C_DIS
LIN {X -0.028,Y -548.549,Z 1121.778,A 0.000,B 0.000,C 90.000,E1 176.045} C_DIS
LIN {X 0.104,Y -555.268,Z 1121.770,A 0.000,B 0.000,C 90.000,E1 174.489} C_DIS
LIN {X 0.002,Y -561.430,Z 1121.762,A 0.000,B 0.000,C 90.000,E1 173.109} C_DIS
LIN {X -0.088,Y -568.158,Z 1121.753,A 0.000,B 0.000,C 90.000,E1 171.602} C_DIS
LIN {X 0.187,Y -574.164,Z 1121.746,A 0.000,B 0.000,C 90.000,E1 170.208} C_DIS
LIN {X -0.226,Y -578.857,Z 1121.740,A 0.000,B 0.000,C 90.000,E1 169.162} C_DIS
LIN {X 0.102,Y -583.353,Z 1121.734,A 0.000,B 0.000,C 90.000,E1 168.049} C_DIS
LIN {X -0.142,Y -589.906,Z 1121.725,A 0.000,B 0.000,C 90.000,E1 166.464} C_DIS
LIN {X 0.183,Y -595.105,Z 1121.717,A 0.000,B 0.000,C 90.000,E1 165.102} C_DIS
LIN {X -0.134,Y -597.988,Z 1121.713,A 0.000,B 0.000,C 90.000,E1 164.338} C_DIS
LIN {X -0.263,Y -600.826,Z 1121.709,A 0.000,B 0.000,C 90.000,E1 163.559} C_DIS
LIN {X -0.160,Y -605.099,Z 1121.701,A 0.000,B 0.000,C 90.000,E1 162.236} C_DIS
LIN {X 0.017,Y -609.214,Z 1121.694,A 0.000,B 0.000,C 90.000,E1 160.913} C_DIS
LIN {X -0.111,Y -613.096,Z 1121.687,A 0.000,B 0.000,C 90.000,E1 159.625} C_DIS
LIN {X 0.144,Y -617.397,Z 1121.678,A 0.000,B 0.000,C 90.000,E1 158.050} C_DIS
LIN {X -0.192,Y -620.807,Z 1121.671,A 0.000,B 0.000,C 90.000,E1 156.794} C_DIS
LIN {X 0.110,Y -624.751,Z 1121.662,A 0.000,B 0.000,C 90.000,E1 155.229} C_DIS
LIN {X -0.067,Y -629.069,Z 1121.653,A 0.000,B 0.000,C 90.000,E1 153.461} C_DIS
LIN {X 0.030,Y -631.438,Z 1121.647,A 0.000,B 0.000,C 90.000,E1 152.436} C_DIS
LIN {X 0.013,Y -635.287,Z 1121.637,A 0.000,B 0.000,C 90.000,E1 150.667} C_DIS
LIN {X -0.008,Y -637.947,Z 1121.630,A 0.000,B 0.000,C 90.000,E1 149.410} C_DIS
LIN {X 0.345,Y -640.457,Z 1121.623,A 0.000,B 0.000,C 90.000,E1 148.122} C_DIS
LIN {X 0.262,Y -643.337,Z 1121.615,A 0.000,B 0.000,C 90.000,E1 146.628} C_DIS
LIN {X -0.246,Y -645.172,Z 1121.609,A 0.000,B 0.000,C 90.000,E1 145.674} C_DIS
LIN {X 0.058,Y -647.277,Z 1121.602,A 0.000,B 0.000,C 90.000,E1 144.402} C_DIS
LIN {X -0.034,Y -649.013,Z 1121.597,A 0.000,B 0.000,C 90.000,E1 143.417} C_DIS
LIN {X 0.165,Y -652.932,Z 1121.584,A 0.000,B 0.000,C 90.000,E1 141.170} C_DIS
LIN {X -0.016,Y -655.172,Z 1121.578,A 0.000,B 0.000,C 90.000,E1 139.952} C_DIS
LIN {X -0.158,Y -658.442,Z 1121.568,A 0.000,B 0.000,C 90.000,E1 138.243} C_DIS
LIN {X 0.196,Y -660.814,Z 1121.561,A 0.000,B 0.000,C 90.000,E1 136.986} C_DIS
LIN {X -0.367,Y -664.398,Z 1121.552,A 0.000,B 0.000,C 90.000,E1 135.324} C_DIS
LIN {X 0.107,Y -669.409,Z 1121.540,A 0.000,B 0.000,C 90.000,E1 133.095} C_DIS
LIN {X 0.248,Y -674.080,Z 1121.529,A 0.000,B 0.000,C 90.000,E1 131.148} C_DIS
LIN {X 0.003,Y -677.540,Z 1121.521,A 0.000,B 0.000,C 90.000,E1 129.725} C_DIS
LIN {X -0.014,Y -682.509,Z 1121.510,A 0.000,B 0.000,C 90.000,E1 127.810} C_DIS
LIN {X 0.390,Y -685.582,Z 1121.503,A 0.000,B 0.000,C 90.000,E1 126.583} C_DIS
LIN {X 0.071,Y -689.103,Z 1121.496,A 0.000,B 0.000,C 90.000,E1 125.185} C_DIS
LIN {X -0.181,Y -692.598,Z 1121.488,A 0.000,B 0.000,C 90.000,E1 123.785} C_DIS
LIN {X -0.033,Y -695.443,Z 1121.481,A 0.000,B 0.000,C 90.000,E1 122.594} C_DIS
LIN {X 0.001,Y -698.071,Z 1121.475,A 0.000,B 0.000,C 90.000,E1 121.416} C_DIS
LIN {X 0.190,Y -699.866,Z 1121.469,A 0.000,B 0.000,C 90.000,E1 120.463} C_DIS
LIN {X 0.249,Y -702.617,Z 1121.460,A 0.000,B 0.000,C 90.000,E1 118.821} C_DIS
LIN {X -0.150,Y -703.800,Z 1121.456,A 0.000,B 0.000,C 90.000,E1 118.153} C_DIS
LIN {X 0.038,Y -704.867,Z 1121.451,A 0.000,B 0.000,C 90.000,E1 117.206} C_DIS
LIN {X -0.012,Y -705.297,Z 1121.449,A 0.000,B 0.000,C 90.000,E1 116.744} C_DIS
LIN {X -0.137,Y -706.050,Z 1121.442,A 0.000,B 0.000,C 90.000,E1 115.591} C_DIS
LIN {X 0.147,Y -706.258,Z 1121.440,A 0.000,B 0.000,C 90.000,E1 115.103} C_DIS
LIN {X 0.091,Y -706.101,Z 1121.437,A 0.000,B 0.000,C 90.000,E1 114.643} C_DIS
LIN {X -0.261,Y -705.374,Z 1121.434,A 0.000,B 0.000,C 90.000,E1 114.207} C_DIS
LIN {X 0.028,Y -704.965,Z 1121.433,A 0.000,B 0.000,C 90.000,E1 113.951} C_DIS
LIN {X -0.329,Y -703.145,Z 1121.431,A 0.000,B 0.000,C 90.000,E1 113.515} C_DIS
LIN {X -0.050,Y -702.005,Z 1121.429,A 0.000,B 0.000,C 90.000,E1 113.259} C_DIS
LIN {X 0.219,Y -697.754,Z 1121.427,A 0.000,B 0.000,C 90.000,E1 112.770} C_DIS
LIN {X 0.349,Y -696.538,Z 1121.426,A 0.000,B 0.000,C 90.000,E1 112.642} C_DIS
LIN {X -0.165,Y -694.662,Z 1121.425,A 0.000,B 0.000,C 90.000,E1 112.567} C_DIS
LIN {X -0.136,Y -686.569,Z 1121.424,A 0.000,B 0.000,C 90.000,E1 112.259} C_DIS
LIN {X -0.134,Y -684.446,Z 1121.423,A 0.000,B 0.000,C 90.000,E1 112.206} C_DIS
LIN {X 0.117,Y -676.595,Z 1121.423,A 0.000,B 0.000,C 90.000,E1 112.099} C_DIS
LIN {X 0.057,Y -603.388,Z 1121.423,A 0.000,B 0.000,C 90.000,E1 112.099} C_DIS
LIN {X -0.077,Y -599.887,Z 1121.422,A 0.000,B 0.000,C 90.000,E1 111.897} C_DIS
LIN {X 0.179,Y -595.489,Z 1121.420,A 0.000,B 0.000,C 90.000,E1 111.535} C_DIS
LIN {X 0.188,Y -580.034,Z 1121.412,A 0.000,B 0.000,C 90.000,E1 110.174} C_DIS
LIN {X 0.085,Y -574.371,Z 1121.410,A 0.000,B 0.000,C 90.000,E1 109.704} C_DIS
LIN {X -0.123,Y -568.369,Z 1121.407,A 0.000,B 0.000,C 90.000,E1 109.268} C_DIS
LIN {X -0.166,Y -561.855,Z 1121.405,A 0.000,B 0.000,C 90.000,E1 108.852} C_DIS
LIN {X 0.038,Y -553.875,Z 1121.402,A 0.000,B 0.000,C 90.000,E1 108.362} C_DIS
LIN {X -0.115,Y -550.194,Z 1121.401,A 0.000,B 0.000,C 90.000,E1 108.109} C_DIS
LIN {X -0.157,Y -549.098,Z 1121.400,A 0.000,B 0.000,C 90.000,E1 107.928} C_DIS
LIN {X 0.323,Y -549.084,Z 1121.400,A 0.000,B 0.000,C 90.000,E1 107.873} C_DIS
LIN {X -0.159,Y -548.789,Z 1121.397,A 0.000,B 0.000,C 90.000,E1 107.511} C_DIS
LIN {X 0.028,Y -550.001,Z 1121.387,A 0.000,B 0.000,C 90.000,E1 105.607} C_DIS
LIN {X -0.009,Y -551.461,Z 1121.376,A 0.000,B 0.000,C 90.000,E1 103.647} C_DIS
LIN {X -0.266,Y -553.133,Z 1121.365,A 0.000,B 0.000,C 90.000,E1 101.715} C_DIS
LIN {X 0.093,Y -555.208,Z 1121.353,A 0.000,B 0.000,C 90.000,E1 99.443} C_DIS
